CASE _diCmdState OF
	0://判断对应指令，是否已经处于完成状态，防止出现重复触发情况	
		_diCmdState := _diCmdState + 1;	
	1://传送力值和速度参数
		IF NOT _aRead_VAR.bExecute//等待最后接收结束
		THEN
			_tonDelay(IN:= TRUE,pt:=T#20MS);
			st_IOData.O_ClampForceSet := rTorqueSet;
			st_IOData.O_ClampSpeedSet := rSpeedSet;	
			st_IOData.O_ClampPosSet := rPosAngleSet;	
			IF _tonDelay.Q
			THEN	
				_aEnableSignal[1] := TRUE;//启动参数数据发送	
				_tonDelay(IN:= FALSE);
				_tonCmdTimeout(in:=FALSE);
				_tonTimeout(in:=FALSE);
				_diCmdState := _diCmdState+1; 
			END_IF
		END_IF		
	2://设置读取参数	
		_tonDelay(IN:= NOT _aEnableSignal[1],PT:=T#200MS);
		_tonCmdTimeout(IN:= _aEnableSignal[1],pt:=T#2S);
		IF _tonDelay.Q
		THEN
			_tonCmdTimeout(in:=FALSE);
			_tonCmdTimeout(in:=FALSE);
			_tonDelay(in:=FALSE);
			_diCmdState := 4; 
		END_IF	
		IF _iSendReceiveState = 999
		THEN
			eErrorID := ERG_20_ERROR.FLT_CLAMPCMD_TIMEOUT;		
			_diCmdState := 100;
		END_IF		
	4://设置读取反馈数据
		_tonCmdTimeout(in:=FALSE);
		_tonDelay(IN:= FALSE);	
		_aEnableSignal[4] := TRUE;//读取状态反馈信息 
		_diCmdState := _diCmdState +1;//转到等待夹取完成 	
	5://等到操作完成
		_tonTimeout(in:=TRUE,pt:=T#10S); 
		_tonCmdTimeout(IN:= TRUE,pt:=T#2S);		
		IF NOT _aEnableSignal[4] //等待读取数据完成
		THEN
			_tonDelay(IN:= TRUE,pt:=T#40MS);
			IF st_IOData.I_ClampState = 0 AND ABS(st_IOData.O_ClampPosSet - st_IOData.I_ClampCurrentPos) <= 0.03 AND //松开位置成功
			   eCmd = ERG_20_CMD.Cmd_Release	//松开指令
			THEN			
				_tonCmdTimeout(in:=FALSE);
				_tonTimeout(in:=FALSE);  
				_diCmdState := 100;
				xComplete := TRUE;
			END_IF		
			IF st_IOData.I_ClampState = 2 AND//夹住物体
				 eCmd = ERG_20_CMD.Cmd_Clamp	//夹紧指令
			THEN			
				_tonCmdTimeout(in:=FALSE);
				_tonTimeout(in:=FALSE);  
				_diCmdState := 100;
				xComplete := TRUE;
			END_IF				
			IF st_IOData.I_ClampState = 2 AND //松开位置的时候，检测是否堵转
       	 eCmd = ERG_20_CMD.Cmd_Release	//松开指令
			THEN	
  			_iNGCount := _iNGCount + 1;		
				IF _iNGCount <= 3
				THEN
				  _tonDelay(IN:=FALSE);
					_diCmdState := _diCmdState + 1;
				ELSE
					_tonCmdTimeout(in:=FALSE);
					_tonTimeout(in:=FALSE);  
					eErrorID := ERG_20_ERROR.FLT_ClAMP_RELEASEFAIL;		
					_diCmdState := 999;
				END_IF				
			END_IF		
			IF st_IOData.I_ClampState = 0 AND ABS(st_IOData.O_ClampPosSet - st_IOData.I_ClampCurrentPos) <= 0.03 AND//没有夹住物体，到位置，判定夹持失败(放个误差数值)
				 eCmd = ERG_20_CMD.Cmd_Clamp	//夹紧指令
			THEN
				_iNGCount := _iNGCount + 1;		
				IF _iNGCount <= 3
				THEN
				  _tonDelay(IN:=FALSE);
					_diCmdState := _diCmdState + 1;
				ELSE
					_tonCmdTimeout(in:=FALSE);
					_tonTimeout(in:=FALSE);  			
					eErrorID := ERG_20_ERROR.FLT_ClAMP_CLAMPFAIL;		
					_diCmdState := 999;
				END_IF
			END_IF	
			IF _tonDelay.Q//做延时刷新
			THEN
				_diCmdState := 4;
			END_IF			
		END_IF
		IF _iSendReceiveState = 999//回原点指令响应超时
		THEN
			eErrorID := ERG_20_ERROR.FLT_CLAMPCMD_TIMEOUT;		
			_diCmdState := 999;
		END_IF
		IF _tonTimeout.Q//回原点动作超时
		THEN
			eErrorID := ERG_20_ERROR.FLT_CLAMP_TIMEOUT;
			_diCmdState := 999;
		END_IF
	6:
		_tonDelay(IN:= TRUE,pt:=T#40MS);
		IF _tonDelay.Q//做延时刷新
		THEN			
			_diCmdState := 0;
		END_IF	
	ELSE
		;	
END_CASE
END_METHOD

METHOD CmdRotateAction
VAR_OUTPUT
	xComplete: BOOL;
END_VAR
// return the real actual fault number
IF eErrorID <> ERG_20_ERROR.NO_ERROR
THEN
  RETURN;  
END_IF
  
IF NOT xRefOk THEN//设备没有原点报警
	eErrorID := ERG_20_ERROR.FLT_xRefOk;
	RETURN;
END_IF

IF rTorqueSet>1 OR rTorqueSet<0.2
	OR rSpeedSet>1440 OR rSpeedSet<1
	OR rPosAngleSet>360000 OR rPosAngleSet<-360000
THEN
	eErrorID := ERG_20_ERROR.FLT_PARA;	
END_IF


CASE _diCmdState OF
	0://判断是否已经处于目标位置或者夹取完成状态，防止出现重复触发情况
		_diCmdState := _diCmdState + 1;
			diOldStep:=_diCmdState;
		_tonDelay(IN:= FALSE);
		IF eCmd = ERG_20_CMD.Cmd_RotateAbsRelease//只有绝对松瓶盖定位是有可能处于目标完成状态的，判断是否已经到目标位置
		THEN
			//检测是否已经处于目标位置
			IF ABS(rPosAngleSet - st_IOData.I_RotateCurrentPos) <= 0.03
			THEN
				_tonTimeout(in:=FALSE);  
				_diCmdState := 100;
				xComplete := TRUE;
			END_IF			
		END_IF
		IF eCmd = ERG_20_CMD.Cmd_RotateAbsClamp//只有绝对定位是有可能处于目标完成状态的，增量的是一定要动作的
		THEN
			//检测是否已经处于目标位置，要是到位置，代表夹紧失败，此时需要报警
			IF ABS(rPosAngleSet - st_IOData.I_RotateCurrentPos) <= 0.03
			THEN
				eErrorID := ERG_20_ERROR.FLT_ROTATE_CLAMPFAIL;
				_diCmdState := 999;
			END_IF
		END_IF
	1://传送参数
			diOldStep:=_diCmdState;
		IF NOT _aRead_VAR.bExecute//等待最后接收结束
		THEN
	    _tonDelay(IN:= TRUE,pt:=T#20MS);//保证执行的都是当次任务 			
			st_IOData.O_RotateForceSet := rTorqueSet;
			st_IOData.O_RotateSpeedSet := rSpeedSet;	
			st_IOData.O_RotatePosSet := rPosAngleSet;				
			IF _tonDelay.Q
			THEN				
				_aEnableSignal[2] := TRUE;//启动旋转绝对定位参数数据发送		    					
				_tonCmdTimeout(in:=FALSE);
				_tonDelay(IN:=FALSE);
				_diCmdState := _diCmdState+1; 	
			END_IF			
		END_IF	
	2://设置读取参数
			diOldStep:=_diCmdState;
		_tonDelay(IN:= NOT _aEnableSignal[2],PT:=T#200MS);//等待设备运行起来
		_tonCmdTimeout(IN:= _aEnableSignal[2],pt:=T#2S);
		IF _tonDelay.Q//等待电动夹爪开始响应
		THEN
			_tonTimeout(in:=FALSE);		
			_diCmdState := _diCmdState +1; 
		END_IF	
		IF _iSendReceiveState = 999//指令执行超时
		THEN
			eErrorID := ERG_20_ERROR.FLT_ROTATECMD_TIMEOUT;		
			_diCmdState := 999;
		END_IF	
	3://设置读取参数反馈
			diOldStep:=_diCmdState;
		_tonCmdTimeout(in:=FALSE);
		_tonDelay(IN:= FALSE);
	  _aEnableSignal[4] := TRUE;   
		_diCmdState := _diCmdState +1;//
	4:
		diOldStep:=_diCmdState;
		_tonTimeout(in:=TRUE,pt:=T#20S); 
		_tonCmdTimeout(IN:= TRUE,pt:=T#2S);
		//进行数据刷新		
		IF NOT _aEnableSignal[4] //等待读取数据完成
		THEN
			_tonDelay(IN:= TRUE,pt:=T#50MS);
			IF ( st_IOData.I_RotateState = 0 ) AND ABS(st_IOData.O_RotatePosSet - st_IOData.I_RotateCurrentPos) <= 0.03 AND //旋转是否到位置,只有在松开瓶盖的时候会有这种操作
				 ( eCmd = ERG_20_CMD.Cmd_RotateAbsRelease )
			THEN			
				_tonTimeout(in:=FALSE);  
				_diCmdState := 100;
				xComplete := TRUE;
			END_IF		 
			IF ( st_IOData.I_RotateState = 2 OR st_IOData.I_RotateState = 4 ) AND //旋转夹瓶盖处理，只有出现堵转（达到设置力反馈）
				 ( eCmd = ERG_20_CMD.Cmd_RotateAbsClamp )
			THEN			
				_tonTimeout(in:=FALSE);  
				_diCmdState := 100;
				xComplete := TRUE;
			END_IF			
			IF _tonDelay.Q//做刷新处理
			THEN
				_diCmdState := _diCmdState - 1;
			END_IF
		END_IF
		IF ( st_IOData.I_RotateState = 0 ) AND ABS(st_IOData.O_RotatePosSet - st_IOData.I_RotateCurrentPos) <= 0.03 AND //关盖打滑,直接到设置位置了
			 ( eCmd = ERG_20_CMD.Cmd_RotateAbsClamp )
		THEN	
			_tonDelay(IN:=FALSE);
			eErrorID := ERG_20_ERROR.FLT_ROTATE_CLAMPFAIL;
			_diCmdState := 999;
		END_IF
		IF ( st_IOData.I_RotateState = 2 OR st_IOData.I_RotateState = 4) AND //开盖失败，直接堵转，开不开瓶盖
			 ( eCmd = ERG_20_CMD.Cmd_RotateAbsRelease )
		THEN	
			_iNGCount := _iNGCount + 1;		
			IF _iNGCount <= 3//检测是否有正时报警发生
			THEN
				_tonDelay(IN:=FALSE);
				_diCmdState := _diCmdState + 1;
			ELSE
				eErrorID := ERG_20_ERROR.FLT_ROTATE_RELEASEFAIL;
				_diCmdState := 999;
			END_IF
		END_IF
		IF _iSendReceiveState = 999//回原点指令响应超时
		THEN
			eErrorID := ERG_20_ERROR.FLT_ROTATECMD_TIMEOUT;		
			_diCmdState := 999;
		END_IF
		IF _tonTimeout.Q//回原点动作超时
		THEN
			eErrorID := ERG_20_ERROR.FLT_ROTATE_TIMEOUT;
			_diCmdState := 999;
		END_IF
	5://报警再次确定
			diOldStep:=_diCmdState;
		_tonDelay(IN:= TRUE,pt:=T#40MS);
		IF _tonDelay.Q//做延时刷新
		THEN			
			_diCmdState := 0;
		END_IF		
	ELSE
		;	
END_CASE
END_METHOD

METHOD CmdRotateAction_Rel
VAR_OUTPUT
	xComplete: BOOL;
END_VAR
// return the real actual fault number
IF eErrorID <> ERG_20_ERROR.NO_ERROR
THEN
  RETURN;  
END_IF
  
IF NOT xRefOk THEN//设备没有原点报警
	eErrorID := ERG_20_ERROR.FLT_xRefOk;
	RETURN;
END_IF

IF rTorqueSet>1 OR rTorqueSet<0.2
	OR rSpeedSet>1440 OR rSpeedSet<1
	OR rPosAngleSet>36000 OR rPosAngleSet<-36000
THEN
	eErrorID := ERG_20_ERROR.FLT_PARA;	
END_IF

CASE _diCmdState OF
	0://判断是否已经处于目标位置或者夹取完成状态，防止出现重复触发情况
		_tonDelay(IN:= FALSE);
		IF NOT _aRead_VAR.bExecute THEN		
			_diCmdState := _diCmdState + 1;
			_rLastRotatePos:= st_IOData.I_RotateCurrentPos;
		END_IF	
	1://传送参数
		_tonDelay(IN:= TRUE,pt:=T#20MS);//保证执行的都是当次任务 			
		st_IOData.O_RotateForceSet := rTorqueSet;
		st_IOData.O_RotateSpeedSet := rSpeedSet;	
		st_IOData.O_RotatePosSet := rPosAngleSet;				
		IF _tonDelay.Q
		THEN				
			_aEnableSignal[3] := TRUE;//启动旋转绝对定位参数数据发送		    					
			_tonCmdTimeout(in:=FALSE);
			_tonDelay(IN:=FALSE);
			_diCmdState := _diCmdState+1; 	
		END_IF			
	2://设置读取参数
		_tonDelay(IN:= NOT _aEnableSignal[3],PT:=T#200MS);//等待设备运行起来
		_tonCmdTimeout(IN:= _aEnableSignal[3],pt:=T#2S);
		IF _tonDelay.Q//等待电动夹爪开始响应
		THEN
			_tonTimeout(in:=FALSE);		
			_diCmdState := _diCmdState +1; 
		END_IF	
		IF _iSendReceiveState = 999//指令执行超时
		THEN
			eErrorID := ERG_20_ERROR.FLT_ROTATECMD_TIMEOUT;		
			_diCmdState := 999;
		END_IF	
	3://设置读取参数反馈
		_tonCmdTimeout(in:=FALSE);
		_tonDelay(IN:= FALSE);
	  _aEnableSignal[4] := TRUE;   
		_diCmdState := _diCmdState +1;//
	4:
		_tonTimeout(in:=TRUE,pt:=T#20S); 
		_tonCmdTimeout(IN:= TRUE,pt:=T#2S);
		//进行数据刷新		
		IF NOT _aEnableSignal[4] //等待读取数据完成
		THEN
			_tonDelay(IN:= TRUE,pt:=T#50MS);
			IF ( st_IOData.I_RotateState = 0 ) 
					AND (st_IOData.I_RotateCurrentPos - _rLastRotatePos) <= rPosAngleSet+0.03 
					AND (st_IOData.I_RotateCurrentPos - _rLastRotatePos) >= rPosAngleSet-0.03 //旋转是否到位置,只有在松开瓶盖的时候会有这种操作
				 AND ( eCmd = ERG_20_CMD.Cmd_RotateRelRelease )
			THEN			
				_tonTimeout(in:=FALSE);  
				_diCmdState := 100;
				xComplete := TRUE;
			END_IF		 
			IF ( st_IOData.I_RotateState = 2 OR st_IOData.I_RotateState = 4 ) AND //旋转夹瓶盖处理，只有出现堵转（达到设置力反馈）
				 ( eCmd = ERG_20_CMD.Cmd_RotateRelClamp )
			THEN			
				_tonTimeout(in:=FALSE);  
				_diCmdState := 100;
				xComplete := TRUE;
			END_IF			
			IF _tonDelay.Q//做刷新处理
			THEN
				_diCmdState := _diCmdState - 1;
			END_IF
		END_IF
		
		IF ( st_IOData.I_RotateState = 0 )  
 				AND (st_IOData.I_RotateCurrentPos - _rLastRotatePos) <= rPosAngleSet+0.03 
				AND (st_IOData.I_RotateCurrentPos - _rLastRotatePos) >= rPosAngleSet-0.03  //关盖打滑,直接到设置位置了
			  AND( eCmd = ERG_20_CMD.Cmd_RotateRelClamp )
		THEN	
			_tonDelay(IN:=FALSE);
			eErrorID := ERG_20_ERROR.FLT_ROTATE_CLAMPFAIL;
			_diCmdState := 999;
		END_IF
		IF ( st_IOData.I_RotateState = 2 OR st_IOData.I_RotateState = 4) AND //开盖失败，直接堵转，开不开瓶盖
			 ( eCmd = ERG_20_CMD.Cmd_RotateRelRelease )
		THEN	
			_iNGCount := _iNGCount + 1;		
			IF _iNGCount <= 3//检测是否有正时报警发生
			THEN
				_tonDelay(IN:=FALSE);
				_diCmdState := _diCmdState + 1;
			ELSE
				eErrorID := ERG_20_ERROR.FLT_ROTATE_RELEASEFAIL;
				_diCmdState := 999;
			END_IF
		END_IF
		IF _iSendReceiveState = 999//回原点指令响应超时
		THEN
			eErrorID := ERG_20_ERROR.FLT_ROTATECMD_TIMEOUT;		
			_diCmdState := 999;
		END_IF
		IF _tonTimeout.Q//回原点动作超时
		THEN
			eErrorID := ERG_20_ERROR.FLT_ROTATE_TIMEOUT;
			_diCmdState := 999;
		END_IF
	5://报警再次确定
		_tonDelay(IN:= TRUE,pt:=T#40MS);
		IF _tonDelay.Q//做延时刷新
		THEN			
			_diCmdState := 3;
		END_IF		
	ELSE
		;	
END_CASE
END_METHOD

ACTION ConnectAction:
(**********************************调用收发功能块**********************************)
//状态反馈功能调用
_aRead_VAR(
	sIPAddr:= stPara.strSlaveIP, 
	nTCPPort:=stPara.iSlavePort , 
	nUnitID:= stPara.bySlaveID, 
	nQuantity:= 18, 
	nMBAddr:= 16#0040, 
	cbLength:= 36, 
	pDestAddr:= ADR(_aFeedbackData), 
	bExecute:= , 
	tTimeout:= T#1S, 
	bBusy=> , 
	bError=> , 
	nErrId=> , 
	cbRead=> );		
	
//指令控制部分	
_aWtirt_VAR[0](
	sIPAddr:= stPara.strSlaveIP,
	nTCPPort:= stPara.iSlavePort, 
	nUnitID:= stPara.bySlaveID, 
	nQuantity:= 1, 
	nMBAddr:= 16#0000, 
	cbLength:= 2, 
	pSrcAddr:= ADR(_aControlData[0,0]), 
	bExecute:= , 
	tTimeout:= T#1S, 
	bBusy=> , 
	bError=> , 
	nErrId=> );	
		
_aWtirt_VAR[1](
	sIPAddr:= stPara.strSlaveIP,
	nTCPPort:= stPara.iSlavePort, 
	nUnitID:= stPara.bySlaveID, 
	nQuantity:= 6, 
	nMBAddr:= 16#0002, 
	cbLength:= 12, 
	pSrcAddr:= ADR(_aControlData[1,0]), 
	bExecute:= , 
	tTimeout:= T#1S, 
	bBusy=> , 
	bError=> , 
	nErrId=> );		
	
_aWtirt_VAR[2](
	sIPAddr:= stPara.strSlaveIP,
	nTCPPort:= stPara.iSlavePort, 
	nUnitID:= stPara.bySlaveID, 
	nQuantity:= 8, 
	nMBAddr:= 16#000A, 
	cbLength:= 16, 
	pSrcAddr:= ADR(_aControlData[2,0]), 
	bExecute:= , 
	tTimeout:= T#1S, 
	bBusy=> , 
	bError=> , 
	nErrId=> );		
	
_aWtirt_VAR[3](
	sIPAddr:= stPara.strSlaveIP,
	nTCPPort:= stPara.iSlavePort, 
	nUnitID:= stPara.bySlaveID, 
	nQuantity:= 8, 
	nMBAddr:= 16#000E, 
	cbLength:= 16, 
	pSrcAddr:= ADR(_aControlData[3,0]), 
	bExecute:= , 
	tTimeout:= T#1S, 
	bBusy=> , 
	bError=> , 
	nErrId=> );	
	
//收发流程管控
CASE _iSendReceiveState OF 
	0:
		_tonDelay2(IN:= FALSE);
		_iChannelIndex:= -1;
		FOR i := 0 TO 5 BY 1//进行读取指令的轮训
		DO
		 IF _aEnableSignal[i]//检测有控制指令发生
		 THEN
			 _iChannelIndex:=i;    
			END_IF 
		END_FOR
		IF _iChannelIndex>=4//有读取反馈指令
		THEN								
			IF NOT _aRead_VAR.bBusy AND NOT _aRead_VAR.bError
			THEN
				_aRead_VAR(bExecute := _aEnableSignal[_iChannelIndex]);
				_iSendReceiveState := 10;	
			ELSIF 
				_aRead_VAR.bError
				THEN
				_iSendReceiveState := 999;												
			END_IF													
		END_IF			
		IF _iChannelIndex>=0 AND _iChannelIndex<=3//有控制触发指令
		THEN		
			IF  NOT _aWtirt_VAR[_iChannelIndex].bBusy AND NOT _aWtirt_VAR[_iChannelIndex].bError 
			THEN
				_aWtirt_VAR[_iChannelIndex](bExecute := _aEnableSignal[_iChannelIndex]);
				_iSendReceiveState := 10;							
			END_IF
		END_IF
		
	10://等待读取响应	
		_tonDelay2(IN:= TRUE,PT:=T#3S);
		IF _tonDelay2.Q//超时
		THEN
			_iSendReceiveState:= 999;					
		END_IF				
		IF _iChannelIndex>=4
		THEN					
			IF NOT _aRead_VAR.bBusy AND NOT _aRead_VAR.bError
			THEN
				_iComNGCount := 0;
				_aEnableSignal[_iChannelIndex] := FALSE;
				_aRead_VAR.bExecute := FALSE;
				_iSendReceiveState := 0;//等待下次触发
			END_IF
			IF _aRead_VAR.bError
			THEN
				_iComNGCount := _iComNGCount + 1;//错误次数加一
				IF _iComNGCount >= 3//重发多次失败
				THEN
					eOperErrorID := _aRead_VAR.nErrId;
					_aRead_VAR.bExecute := FALSE;
					_iSendReceiveState := 999;//进入错误发生状态
				ELSE
					_tonDelay1(in:=FALSE);
					_aRead_VAR.bExecute:= FALSE;
					_iSendReceiveState := _iSendReceiveState + 1;
				END_IF						
			END_IF			
		END_IF				
		IF _iChannelIndex>=0 AND _iChannelIndex<=3		
		THEN	
			IF NOT _aWtirt_VAR[_iChannelIndex].bBusy AND NOT _aWtirt_VAR[_iChannelIndex].bError
			THEN
				_iComNGCount := 0;
				_aEnableSignal[_iChannelIndex] := FALSE;
				_aWtirt_VAR[_iChannelIndex].bExecute := FALSE;
				_iSendReceiveState := 0;//等待下次触发
			END_IF
			IF _aWtirt_VAR[_iChannelIndex].bError
			THEN
				_iComNGCount := _iComNGCount + 1;//错误次数加一
				IF _iComNGCount >= 3//重发多次失败
				THEN
					eOperErrorID := _aWtirt_VAR[_iChannelIndex].nErrId;
					_aWtirt_VAR[_iChannelIndex].bExecute := FALSE;
					_iSendReceiveState := 999;//进入错误发生状态
				ELSE
					_tonDelay1(in:=FALSE);
					_aWtirt_VAR[_iChannelIndex].bExecute:= FALSE;
					_iSendReceiveState := _iSendReceiveState + 1;
				END_IF					
			END_IF				
		END_IF
	11://延时，进行补发操作
		_tonDelay1(in:=TRUE,pt:=T#300MS);				
		IF _tonDelay1.Q
		THEN		 
			_iSendReceiveState := 0;
		END_IF	
	999://错误状态，等待复位发生
		_xConnect_ERROR := TRUE;
		_tonDelay1(in:=NOT _tonDelay1.Q,pt:=T#20MS);
		_aRead_VAR(bExecute := _tonDelay1.Q);	
		_tonDelay3(pt:=T#100MS);	
		IF _tonDelay3.Q
		THEN			
			_xConnect_ERROR := FALSE;
			_iComNGCount := 0;			
			_iSendReceiveState := 0;//重新开始
			_aRead_VAR(bExecute := FALSE);	
			_tonDelay1(IN:=FALSE);
			_tonDelay3(IN:=FALSE);
		END_IF
		IF _fResetCheck.Q
		THEN
			_aWtirt_VAR[0](bExecute := FALSE);
			_aWtirt_VAR[1](bExecute := FALSE);
			_aWtirt_VAR[2](bExecute := FALSE);
			_aWtirt_VAR[3](bExecute := FALSE);			
			_aRead_VAR(bExecute := FALSE);	
			_tonDelay3.IN := TRUE;
		END_IF
	ELSE
		;
END_CASE
END_ACTION

METHOD CyclicAction
VAR_INPUT
END_VAR
VAR_OUTPUT
	xComplete: BOOL;
END_VAR
IF xAbort=0 THEN
    IF xFirstInvocation THEN
    (*
    * Staring
    * for then first (!) invocaion,
    * sample then input variables
    *)
			_xReadStatus := FALSE;
			_iCount := 0;
			_diCmdState := 0;
			_iNGCount := 0;
			xFirstInvocation:=0;	
			_aRead_VAR.bExecute:= false;		
    END_IF    
    REPEAT 				
		  (**************************检查是否有硬件报错(检测总线是否报错)**********************************) 			
			//下面几个报警需要断驱动器的电才能消除报警
			IF st_IOData.I_DeviceERRORState <> 0 
			THEN
				eErrorID := ERG_20_ERROR.FLT_DEVICE_ERROR;//过热报警
			END_IF	

			IF NOT xPowerHmi//驱动器没有上电
			THEN
				eERRORID := ERG_20_ERROR.FLT_POWERON;//需要检查硬件，硬件有问题
			END_IF
		
			//判断指令类型
			CASE eCmd OF
					ERG_20_CMD.Cmd_Clamp,ERG_20_CMD.Cmd_Release://执行夹爪指令	
            eClampActCmd := eCmd ;				
						CmdClampAction(xComplete=> xComplete);				
					ERG_20_CMD.Cmd_Org://执行回原点指令
						mCmdOrgAction(xComplete=> xComplete);
					ERG_20_CMD.Cmd_RotateAbsClamp,ERG_20_CMD.Cmd_RotateAbsRelease:
						CmdRotateAction(xComplete=> xComplete);
					ERG_20_CMD.Cmd_RotateRelClamp,ERG_20_CMD.Cmd_RotateRelRelease:
						CmdRotateAction_Rel(xComplete=> xComplete);												
					ELSE
						;	
				END_CASE  
      UNTIL (TRUE)
	END_REPEAT
END_IF


IF xAbort OR xComplete OR eErrorID<>ERG_20_ERROR.NO_ERROR THEN    
    (*
    * Cleaning
    * => free as much allocated resources as possible
    *)    
    tOperationTimer(IN:=0);
END_IF
END_METHOD

{attribute 'hide'}
METHOD PRIVATE FINAL HandleAbortedState
VAR_INPUT
END_VAR
VAR_OUTPUT
	xAgain: BOOL;
END_VAR
VAR
	xComplete: BOOL;
END_VAR
IF xAborted AND xResetRequest THEN
    eState:=STATE.RESETING;
    xAgain:=1;
ELSE
    xBusy:=0;
    xAborted:=1;
    //xResetRequest:=(xExecute=0);
    xAgain:=0;(* !!! *)
END_IF
END_METHOD

{attribute 'hide'}
METHOD PRIVATE FINAL HandleAbortingState
VAR_INPUT
END_VAR
VAR_OUTPUT
	xAgain: BOOL;
END_VAR
VAR
	xComplete: BOOL;
END_VAR
AbortAction(xComplete=> xComplete, eErrorID=> eErrorID);

IF eErrorID<>ERG_20_ERROR.NO_ERROR THEN
    eState:=STATE.INERROR;
    xAgain:=1;
ELSIF xComplete THEN
    eState:=STATE.ABORTED;
    xAgain:=1;
END_IF
END_METHOD

{attribute 'hide'}
METHOD PRIVATE FINAL HandleDoneState
VAR_INPUT
END_VAR
VAR_OUTPUT
	xAgain: BOOL;
END_VAR
//在运行过程中要是切换模式，再运行完成之后，检测到模式的切换，就需要回到初始位置，进行下一次执行准备
IF _xDone AND ((xExecute=0) OR ( _xModeChange AND NOT _xAutoOpe ) OR ( NOT xAutoMode AND NOT xDeviceRunning AND ( NOT _xAutoOpe OR _xHMIOpe))) THEN
	eState:=STATE.RESETING;
	xAgain:=1;
ELSE
	xBusy:=0;
	_xDone:=1;
	//xResetRequest:=(xExecute=0);
	xAgain:=0;(* !!! *)
END_IF
END_METHOD

{attribute 'hide'}
METHOD PRIVATE FINAL HandleDormantState
VAR_INPUT
END_VAR
VAR_OUTPUT
	xAgain: BOOL;
END_VAR

IF xExecute THEN
    xBusy:=1;
    eState:=STATE.EXECUTING;
    xAgain:=1;
END_IF


IF st_IOData.I_DeviceERRORState <> 0//检测硬件是否报错
THEN
	eERRORID := ERG_20_ERROR.FLT_DEVICE_ERROR;//需要检查硬件，硬件有问题
END_IF
IF NOT xPowerHmi//驱动器没有上电
THEN
	eERRORID := ERG_20_ERROR.FLT_POWERON;//需要检查硬件，硬件有问题
END_IF
	
IF _fResetCheck.Q//清空报警
THEN
	eERRORID := ERG_20_ERROR.No_ERROR;
END_IF
(********************************等待手动操作******************************)
//初始化指令
_rHMIInit(CLK:= xHMInitButton AND eErrorID = ERG_20_ERROR.NO_ERROR AND NOT xAutoMode AND NOT xDeviceRunning );
_rInit(CLK:= xInitControl AND eErrorID = ERG_20_ERROR.NO_ERROR AND ( xAutoMode OR  xDeviceRunning ));
IF _rHMIInit.Q OR _rInit.Q
THEN
	eCmd := ERG_20_CMD.Cmd_Org;
	xExecute := TRUE;
END_IF
//轮询
FOR ii := 1 TO 5 BY 1
DO 
	//夹紧轴夹紧控制
	_rHMIClamp[ii](CLK:= aHMIClampButton[ii] AND eErrorID = ERG_20_ERROR.NO_ERROR AND NOT xAutoMode AND NOT xDeviceRunning );
	_rClamp[ii](CLK:= aClampControl[ii] AND eErrorID = ERG_20_ERROR.NO_ERROR AND ( xAutoMode OR xDeviceRunning ) );
	IF _rHMIClamp[ii].Q OR _rClamp[ii].Q
	THEN
		rTorqueSet := aHMIClampPara[ii].rTorqueSet;
		rSpeedSet := aHMIClampPara[ii].rSpeedSet;
		rPosAngleSet := aHMIClampPara[ii].rPosAngleSet;
		eCmd := ERG_20_CMD.Cmd_Clamp;
		xExecute := TRUE;
	END_IF	
	//夹紧轴松开指令
	_rHMIRelease[ii](CLK:= aHMIReleaseButton[ii] AND eErrorID = ERG_20_ERROR.NO_ERROR AND NOT xAutoMode AND NOT xDeviceRunning );
	_rRelease[ii](CLK:= aReleaseControl[ii] AND eErrorID = ERG_20_ERROR.NO_ERROR AND ( xAutoMode OR  xDeviceRunning ));
	IF _rHMIRelease[ii].Q OR _rRelease[ii].Q
	THEN
		rTorqueSet := aHMIReleasePara[ii].rTorqueSet;
		rSpeedSet := aHMIReleasePara[ii].rSpeedSet;
		rPosAngleSet := aHMIReleasePara[ii].rPosAngleSet;
		eCmd := ERG_20_CMD.Cmd_Release;
		xExecute := TRUE;
	END_IF		
  //旋转轴关盖控制
	_rHMIRotateClamp[ii](CLK:= aHMIRotateClampButton[ii] AND eErrorID = ERG_20_ERROR.NO_ERROR AND NOT xAutoMode AND NOT xDeviceRunning );
	_rRotateClamp[ii](CLK:= aRotateClampControl[ii] AND eErrorID = ERG_20_ERROR.NO_ERROR AND ( xAutoMode OR xDeviceRunning ) );
	IF _rHMIRotateClamp[ii].Q OR _rRotateClamp[ii].Q
	THEN
		rTorqueSet := aHMIRotateClampPara[ii].rTorqueSet;
		rSpeedSet := aHMIRotateClampPara[ii].rSpeedSet;
		rPosAngleSet := aHMIRotateClampPara[ii].rPosAngleSet;
		eCmd := ERG_20_CMD.Cmd_RotateAbsClamp;
		xExecute := TRUE;
	END_IF	
	//旋转轴松盖指令
	_rHMIRotateRelease[ii](CLK:= aHMIRotateReleaseButton[ii] AND eErrorID = ERG_20_ERROR.NO_ERROR AND NOT xAutoMode AND NOT xDeviceRunning );
	_rRotateRelease[ii](CLK:= aRotateReleaseControl[ii] AND eErrorID = ERG_20_ERROR.NO_ERROR AND ( xAutoMode OR  xDeviceRunning ));
	IF _rHMIRotateRelease[ii].Q OR _rRotateRelease[ii].Q
	THEN
		rTorqueSet := aHMIRotateReleasePara[ii].rTorqueSet;
		rSpeedSet := aHMIRotateReleasePara[ii].rSpeedSet;
		rPosAngleSet := aHMIRotateReleasePara[ii].rPosAngleSet;
		eCmd := ERG_20_CMD.Cmd_RotateAbsRelease;
		xExecute := TRUE;
	END_IF		
  //旋转轴关盖控制
	_rHMIRotateRelClamp[ii](CLK:= aHMIRotateClampRelButton[ii] AND eErrorID = ERG_20_ERROR.NO_ERROR AND NOT xAutoMode AND NOT xDeviceRunning );
	_rRotateRelClamp[ii](CLK:= aRotateClampRelControl[ii] AND eErrorID = ERG_20_ERROR.NO_ERROR AND ( xAutoMode OR xDeviceRunning ) );
	IF _rHMIRotateRelClamp[ii].Q OR _rRotateRelClamp[ii].Q
	THEN
		rTorqueSet := aHMIRotateClampRelPara[ii].rTorqueSet;
		rSpeedSet := aHMIRotateClampRelPara[ii].rSpeedSet;
		rPosAngleSet := aHMIRotateClampRelPara[ii].rPosAngleSet;
		eCmd := ERG_20_CMD.Cmd_RotateRelClamp;
		xExecute := TRUE;
	END_IF	
	//旋转轴松盖指令
	_rHMIRotateRelRelease[ii](CLK:= aHMIRotateReleaseRelButton[ii] AND eErrorID = ERG_20_ERROR.NO_ERROR AND NOT xAutoMode AND NOT xDeviceRunning );
	_rRotateRelRelease[ii](CLK:= aRotateReleaseRelControl[ii] AND eErrorID = ERG_20_ERROR.NO_ERROR AND ( xAutoMode OR  xDeviceRunning ));
	IF _rHMIRotateRelRelease[ii].Q OR _rRotateRelRelease[ii].Q
	THEN
		rTorqueSet := aHMIRotateReleaseRelPara[ii].rTorqueSet;
		rSpeedSet := aHMIRotateReleaseRelPara[ii].rSpeedSet;
		rPosAngleSet := aHMIRotateReleaseRelPara[ii].rPosAngleSet;
		eCmd := ERG_20_CMD.Cmd_RotateRelRelease;
		xExecute := TRUE;
	END_IF
END_FOR
END_METHOD

{attribute 'hide'}
METHOD PRIVATE FINAL  HandleErrorState
VAR_INPUT
END_VAR
VAR_OUTPUT
	xAgain: BOOL;
END_VAR
IF xError THEN
	IF eErrorID < ERG_20_ERROR.FLT_ClAMP_CLAMPFAIL//正常执行报警
	THEN
		IF xResetRequest OR NOT xExecute//按照正常逻辑进行处理复位处理就可以
		THEN
				eState:=STATE.RESETING;
				xAgain:=1;
		END_IF
	ELSE//操作失败报警（有可能需要进行程序跳步处理，此时，在自动模式下不允许被复位掉，防止，程序异常死机）
		IF ( NOT xAutoMode AND xDeviceRunning ) OR xAutoMode
		THEN 
			IF NOT xExecute//按照正常逻辑进行处理复位处理就可以
			THEN 
				eState:=STATE.RESETING;
				xAgain:=1;
			END_IF
		ELSE
			IF xResetRequest OR NOT xExecute//按照正常逻辑进行处理复位处理就可以
			THEN
				eState:=STATE.RESETING;
				xAgain:=1;
			END_IF
		END_IF
	END_IF
ELSE
	xBusy:=0;
	xError:=1;    
	xAgain:=0;(* !!! *)
END_IF
END_METHOD

{attribute 'hide'}
METHOD PRIVATE FINAL HandleExecutingState
VAR_INPUT
END_VAR
VAR_OUTPUT
	xAgain: BOOL;
END_VAR
VAR
	xComplete: BOOL;
END_VAR
IF xAbort=0 THEN   
    CyclicAction(xComplete=> xComplete);
END_IF

IF eErrorID<>ERG_20_ERROR.NO_ERROR THEN
    eState:=STATE.INERROR;
    xAgain:=1;
ELSIF xAbort THEN
    eState:=STATE.ABORTING;
    xAgain:=1;
ELSIF xComplete THEN
    eState:=STATE.DONE;
    xAgain:=1;
END_IF
END_METHOD

{attribute 'hide'}
METHOD PRIVATE FINAL HandleResettingState
VAR_INPUT
END_VAR
VAR_OUTPUT
	xAgain: BOOL;
END_VAR
VAR
	xComplete: BOOL;
END_VAR
ResetAction(xComplete=> xComplete);

IF xComplete THEN
		xExecute:=0;//清除输入指令 
    xBusy:=0;
    _xDone:=0;
    xError:=0;
    xAborted:=0;
    eErrorID:=ERG_20_ERROR.NO_ERROR;
    eState:=STATE.DORMANT;
    xFirstInvocation:=1;
    xAgain:=0;(* !!! *)
END_IF
END_METHOD

METHOD mCmdOrgAction
VAR_OUTPUT
	xComplete: BOOL;
END_VAR
// return the real actual fault number
IF eErrorID <> ERG_20_ERROR.NO_ERROR
THEN
  RETURN;  
END_IF

CASE _diCmdState OF
	0://a相关数据初始化
		IF NOT _aRead_VAR.bExecute//等待接收结束
		THEN			
			xRefOk := FALSE;//因为需要重新初始化，所以需要清除回原点完成标志位	
			_aFeedbackData[0]:=0;    
			_diCmdState := _diCmdState+1;						
		END_IF
	1://首次初始化写入参数
			_tonDelay(in:=FALSE);
			_tonCmdTimeout(in:=FALSE);
			_diCmdState:= 2;		
	2://a相关数据初始化
		IF NOT _aRead_VAR.bExecute//等待接收结束
		THEN
			_tonDelay(IN:= TRUE,pt:=T#20MS);
			st_IOData.O_Init := 1;//触发回原点指令
			IF _tonDelay.Q//错开刷新时序
			THEN
				_aEnableSignal[0] := TRUE;//启动数据发送	  
				_tonTimeout(in:=FALSE);    
				_diCmdState := _diCmdState+1;
			END_IF			
		END_IF	
	3://检测指令是否超时
		_tonDelay(IN:= NOT _aEnableSignal[0],PT:=T#200MS);
		_tonCmdTimeout(IN:= _aEnableSignal[0],pt:=T#2S);
		IF _tonDelay.Q
		THEN
			_tonCmdTimeout(in:=FALSE);
			_tonDelay(in:=FALSE);
			_diCmdState := _diCmdState+1; 
		END_IF	
		IF _iSendReceiveState = 999
		THEN
			eErrorID := ERG_20_ERROR.FLT_ORGCMD_TIMEOUT;		
			_diCmdState := 999;
		END_IF		
	4://设置读取数据反馈	 
		_tonCmdTimeout(in:=FALSE);
		_tonTimeout(in:=TRUE,pt:=T#10S); 
		_tonDelay(IN:= FALSE);
		_aEnableSignal[4]:= TRUE;//读取状态信息
		_diCmdState := _diCmdState +1; 
	5://等待数据接收完成		
		_tonTimeout(in:=TRUE,pt:=T#10S); 
		_tonCmdTimeout(IN:= TRUE,pt:=T#2S);
		IF NOT _aEnableSignal[4]//等待电动夹爪响应 
		THEN
			_tonDelay(IN:= TRUE,pt:=T#40MS);
			IF st_IOData.I_ClampInit = 5  //判断是否初始化成功
			THEN
				_tonCmdTimeout(in:=FALSE);
				_tonDelay(IN:= FALSE);
				_tonTimeout(in:=FALSE);  
				_diCmdState := 100;
				xRefOk := TRUE;//标记回原点成功
				xComplete := 1;
			END_IF
			IF _tonDelay.Q
			THEN
				_diCmdState := 4;
			END_IF
		END_IF
		IF _iSendReceiveState = 999//回原点指令响应超时
		THEN
			eErrorID := ERG_20_ERROR.FLT_ORGCMD_TIMEOUT;		
			_diCmdState := 999;
		END_IF
		IF _tonTimeout.Q//回原点动作超时
		THEN
			eErrorID := ERG_20_ERROR.FLT_ORG_TIMEOUT;
			_diCmdState := 999;
		END_IF			
	ELSE
		;
END_CASE
END_METHOD

{attribute 'hide'}
METHOD ResetAction
VAR_INPUT
END_VAR
VAR_OUTPUT
	xComplete: BOOL;
END_VAR
(*
* Cleaning
* => free all allocated resources
* => reinitialize instance variables
*)
tOperationTimer(IN:=0);

// init command state
_diCmdState := 0;
_tonCmdTimeout(in:=FALSE);
_tonTimeout(in:=FALSE);
_tonDelay(IN:=FALSE);
_xModeChange := FALSE;
_iNGCount := 0;
_xReadStatus := TRUE;//操作完成之后，默认开始群进行读取操作

//清除触发标志位
FOR i:= 0 TO 4 BY 1
DO
	_aEnableSignal[i] := FALSE;
END_FOR

xHMInitButton:=FALSE;	
xInitControl:=FALSE;
FOR i:=1 TO 5 BY 1
DO
	aHMIClampButton[i]:=FALSE;
	aHMIReleaseButton[i]:=FALSE;
	aClampControl[i]:=FALSE;
	aReleaseControl[i]:=FALSE;
	aHMIRotateClampButton[i]:=FALSE;
	aHMIRotateReleaseButton[i]:=FALSE;
	aRotateClampControl[i]:=FALSE;
	aRotateReleaseControl[i]:=FALSE;
	
	aHMIRotateClampRelButton[i]:=FALSE;
	aHMIRotateReleaseRelButton[i]:=FALSE;
	aRotateClampRelControl[i]:=FALSE;
	aRotateReleaseRelControl[i]:=FALSE;
END_FOR

xComplete:=1;
END_METHOD

END_FUNCTION_BLOCK

// ---- POUs/003_FB/0014_HITBOT/FB_ERG_20C.TcPOU
FUNCTION_BLOCK FB_ERG_20C EXTENDS FB_Modbus_Tcp
(*
********************************************************************************
* Name: FB_ERG_20C
*
* Author:  Automanh
* Version: 1.0.0
*
* Description:
*  HITBOT's Z_ERG_20C AutoClamp of Rotate and Holding
*  
*
* Remarks:
*
* Revisions:
*   1.0.0 -AutomanH Rebuild
*********************************************************************************)
VAR_INPUT
	xIReset:BOOL;
	xIManualMode:BOOL;
	xIAutoMode:BOOL;
	xIDeviceRunning:BOOL;
	xITryRun:BOOL;//空跑
	LocalClient:stModbusPara;
	stRunPara	:stSetPara;//运行参数	
	stDeviceOpe	:stOper_Para;//操作按钮
END_VAR
VAR_OUTPUT
	stDevice:stDeviceStatus;
	stPara:stDeviceStatus;
	stReadPara:stReadPara;
	iQErrorID:INT;
	strQErrorID:STRING;
END_VAR
VAR
	// 按钮输入
	OperR_TRIG: ARRAY[1..40] OF  R_TRIG;
	//本地参数
	stLocalPara:stHIBOTLocalPara;
	//操作指令
	iOperType:INT;
	// 循环用
	i: INT;
	// //操作类型计数
	iOperCounter: INT;
	// 步骤
	iRunStep,iOldRunStep: INT;
	iParaStep,iOldParaStep:INT;
	// 临时变量
	arwSetData: ARRAY[1..2] OF WORD;
	// 超时定时器
	tTimeout: ARRAY[1..5] OF TON;
	rTempData:REAL;//临时
END_VAR

MEMCPY(ADR(SUPER^.stModbusPara),ADR(LocalClient),SIZEOF(localClient));
SUPER^.M_Modbus();
ACT_Operation();
ACT_Running();
ACT_ERROR();
ACT_Reset();

ACTION ACT_ERROR:
tTimeout[1](IN:= iParaStep =iOldParaStep AND iParaStep<>0 , PT:= T#15S, Q=> , ET=> );
tTimeout[2](IN:= iRunStep =iOldRunStep AND iRunStep<>0 , PT:= T#15S, Q=> , ET=> );
IF		tTimeout[1].Q THEN
	  	stPara.xQError:=TRUE;
	  	stPara.xQBusy:=FALSE;
			iQErrorID:=HITBOT_ERROR.FLT_CMD_TIMEOUT;
	    iParaStep := 999;
END_IF

IF		tTimeout[2].Q THEN
			stDevice.xQError:=TRUE;
			stDevice.xQBusy:=FALSE;
			iQErrorID:=HITBOT_ERROR.FLT_CMD_TIMEOUT;
			iRunStep := 999;
END_IF

IF  iQErrorID<> HITBOT_ERROR.NO_ERROR  THEN
		stDevice.xQError:=TRUE;
END_IF
//报错内容输出
CASE iQErrorID OF 
		 HITBOT_ERROR.No_ERROR:
			 strQErrorID:='NO ERROR';
		 HITBOT_ERROR.FLT_PARA:
			 strQErrorID:='FLT_PARA';
		 HITBOT_ERROR.FLT_READ_PARA:
			 strQErrorID:='FLT_READ_PARA';
		 HITBOT_ERROR.FLT_SET_PARA:
			 strQErrorID:='FLT_SET_PARA';	
		 HITBOT_ERROR.FLT_CMD_TIMEOUT:
			 strQErrorID:='FLT_CMD_TIMEOUT';	
		 HITBOT_ERROR.FLT_RUN_ERROR:
			 strQErrorID:='FLT_RUN_ERROR';	
		 HITBOT_ERROR.FLT_CONFIGURE_PARA:
			 strQErrorID:='FLT_CONFIGURE_PARA';		
		 HITBOT_ERROR.FLT_NEED_INIT:
			 strQErrorID:='FLT_NEED_INIT';	
		 HITBOT_ERROR.FLT_CLAMP_EMPTY:
			strQErrorID:='FLT_CLAMP_EMPTY';		
END_CASE
END_ACTION

ACTION ACT_Operation:
FOR i:=1 TO 5 BY 1 DO
		OperR_TRIG[i](CLK:= (xIManualMode AND  stDeviceOpe.aHMIClampButton[i]) OR((xIAutoMode OR  xIDeviceRunning) AND stDeviceOpe.aClampControl[i]) , Q=> );	//夹紧
END_FOR
FOR i:=6 TO 10 BY 1DO
		OperR_TRIG[i](CLK:= (xIManualMode AND  stDeviceOpe.aHMIReleaseButton[i-5]) OR((xIAutoMode OR  xIDeviceRunning) AND stDeviceOpe.aReleaseControl[i-5]) , Q=> );	//松开
END_FOR
FOR i:=11 TO 15 BY 1 DO
		OperR_TRIG[i](CLK:= (xIManualMode AND  stDeviceOpe.aHMIRotateClampButton[i-10]) OR((xIAutoMode OR  xIDeviceRunning) AND stDeviceOpe.aRotateClampControl[i-10]) , Q=> );	//旋转拧紧
END_FOR

FOR i:=16 TO 20 BY 1 DO
		OperR_TRIG[i](CLK:= (xIManualMode AND  stDeviceOpe.aHMIRotateReleaseButton[i-15]) OR((xIAutoMode OR  xIDeviceRunning) AND stDeviceOpe.aRotateReleaseControl[i-15]) , Q=> );	//旋转松开
END_FOR

FOR i:=21 TO 25 BY 1 DO
		OperR_TRIG[i](CLK:= (xIManualMode AND  stDeviceOpe.aHMIRotateClampRelButton[i-20]) OR((xIAutoMode OR  xIDeviceRunning) AND stDeviceOpe.aRotateClampRelControl[i-20]) , Q=> );	//旋转拧紧-相对
END_FOR

FOR i:=26 TO 30 BY 1 DO
		OperR_TRIG[i](CLK:= (xIManualMode AND  stDeviceOpe.aHMIRotateReleaseRelButton[i-25]) OR((xIAutoMode OR  xIDeviceRunning) AND stDeviceOpe.aRotateReleaseRelControl[i-25]) , Q=> );	//旋转松开-相对
END_FOR
OperR_TRIG[31](CLK:= (xIManualMode AND  stDeviceOpe.xHMInitButton) OR((xIAutoMode OR  xIDeviceRunning) AND stDeviceOpe.xInitControl) , Q=> );	//初始化

FOR  i:= 1 TO 40 BY 1 DO
 	IF   OperR_TRIG[i].Q THEN
				iOperCounter:= i;
				stDevice.xQStart:=TRUE;
				EXIT;
	END_IF
END_FOR
//夹紧
FOR  i:=1 TO 5 BY 1 DO
 		IF   iOperCounter =i THEN
		 		stLocalPara.stClampPara.rPositionSet:=stRunPara.aHMIClampPara[i].rPositionSet;
				stLocalPara.stClampPara.rSpeedSet:=stRunPara.aHMIClampPara[i].rSpeedSet;
				stLocalPara.stClampPara.rCurrentSet:=stRunPara.aHMIClampPara[i].rCurrentSet;
				iOperType:=stCmdType.iClamp;
		END_IF
END_FOR
//松开
FOR  i:=6 TO 10 BY 1 DO
		IF   iOperCounter =i THEN
		 		stLocalPara.stClampPara.rPositionSet:=stRunPara.aHMIReleasePara[i-5].rPositionSet;
				stLocalPara.stClampPara.rSpeedSet:=stRunPara.aHMIReleasePara[i-5].rSpeedSet;
				stLocalPara.stClampPara.rCurrentSet:=stRunPara.aHMIReleasePara[i-5].rCurrentSet;
				iOperType:=stCmdType.iRelease;
		END_IF
END_FOR 
 //拧紧
FOR  i:=11 TO 15 BY 1 DO
 		IF   iOperCounter =i THEN
		 		stLocalPara.stRotateClampPara.rPositionSet:=stRunPara.aHMIRotateClampPara[i-10].rPositionSet;
				stLocalPara.stRotateClampPara.rSpeedSet:=stRunPara.aHMIRotateClampPara[i-10].rSpeedSet;
				stLocalPara.stRotateClampPara.rCurrentSet:=stRunPara.aHMIRotateClampPara[i-10].rCurrentSet;
				iOperType:=stCmdType.iRotateClamp;
		END_IF
END_FOR
//拧松
FOR  i:=16 TO 20 BY 1 DO
		IF   iOperCounter =i THEN
		 		stLocalPara.stRotateClampPara.rPositionSet:=stRunPara.aHMIRotateReleasePara[i-15].rPositionSet;
				stLocalPara.stRotateClampPara.rSpeedSet:=stRunPara.aHMIRotateReleasePara[i-15].rSpeedSet;
				stLocalPara.stRotateClampPara.rCurrentSet:=stRunPara.aHMIRotateReleasePara[i-15].rCurrentSet;
				iOperType:=stCmdType.iRotateRelease;
		END_IF
END_FOR 
 //相对拧紧
FOR  i:=21 TO 26 BY 1 DO
 		IF   iOperCounter =i THEN
		 		stLocalPara.stRotateClampPara.rPositionSet:=stRunPara.aHMIRotateRelClampPara[i-20].rPositionSet;
				stLocalPara.stRotateClampPara.rSpeedSet:=stRunPara.aHMIRotateRelClampPara[i-20].rSpeedSet;
				stLocalPara.stRotateRelAngle:=stRunPara.aHMIRotateRelClampPara[i-20].rCurrentSet;
				iOperType:=stCmdType.iRotateRelClamp;
		END_IF
END_FOR
//相对拧松
FOR  i:=26 TO 30 BY 1 DO
		IF   iOperCounter =i THEN
		 		stLocalPara.stRotateClampPara.rPositionSet:=stRunPara.aHMIRotateRelReleasePara[i-25].rPositionSet;
				stLocalPara.stRotateClampPara.rSpeedSet:=stRunPara.aHMIRotateRelReleasePara[i-25].rSpeedSet;
				stLocalPara.stRotateRelAngle:=stRunPara.aHMIRotateRelReleasePara[i-25].rCurrentSet;
				iOperType:=stCmdType.iRotateRelRelease;
		END_IF
END_FOR 

	IF   iOperCounter =31 THEN
				iOperType:=stCmdType.iInit;
	END_IF


MEMSET(ADR(stDeviceOpe),0,SIZEOF(stDeviceOpe));
END_ACTION

ACTION ACT_Para_Clamp:
CASE iParaStep OF	
	0://开始
			IF   stPara.xQStart THEN
			 		 stPara.xQStart:=FALSE;
					 stPara.xQBusy:=TRUE;
					 stPara.xQDone:=FALSE;
					  iParaStep := iParaStep + 1;
			 END_IF
 	1://查看夹爪电流，转速，转矩
			iOldParaStep:=iParaStep;
			IF 	(stLocalPara.stClampPara.rSpeedSet >=1  	AND 
			 		stLocalPara.stClampPara.rSpeedSet <=1000  )	AND
					(stLocalPara.stClampPara.rPositionSet >=0  AND 
					 stLocalPara.stClampPara.rPositionSet <= 20  )AND 
					(stLocalPara.stClampPara.rCurrentSet >=0.1  AND 
					 stLocalPara.stClampPara.rCurrentSet <=0.5  ) THEN
						iParaStep := iParaStep + 1;	
			ELSE
			 				iQErrorID :=HITBOT_ERROR.FLT_PARA;		
							iParaStep := 999;
			END_IF
	2://读取夹持速度和夹持电流
			iOldParaStep:=iParaStep;
			wMBAddReadRegs:=16#0004;
			wQuantityReadRegs:=4;
			xReadRegs:=TRUE;
			IF  fbReadRegs.bBusy THEN
			 	xReadRegs:=FALSE;
				iParaStep:=iParaStep+1;
			END_IF
	3://等待读取完成
			 	iOldParaStep:=iParaStep;
	  	  IF  NOT 	fbReadRegs.bBusy AND  NOT  	fbReadRegs.bError THEN
				 				//夹持速度
				
								stReadPara.rClampSpeed:=M_Little_Endian(pInputData:=ADR(arwDataReadRegs[1]));
								//夹持电流
						
								stReadPara.rClampCurrent:=M_Little_Endian(pInputData:=ADR(arwDataReadRegs[3]));
	  		 				 iParaStep:=iParaStep+1;
	  		 ELSIF   	fbReadRegs.bError THEN
	  		 			iParaStep:=999;				
	  		 			iQErrorID:=HITBOT_ERROR.FLT_READ_PARA;					
	  		 END_IF	
	4://夹持速度
				iOldParaStep:=iParaStep;
				IF stLocalPara.stClampPara.rSpeedSet <> stReadPara.rClampPosition THEN 
					 iParaStep:=iParaStep + 1;	
				ELSE
					 iParaStep:=iParaStep +4;
				END_IF
	5://夹持速度赋值
			iOldParaStep:=iParaStep;
			MEMCPY(ADR(arwSetData[1]),ADR(stLocalPara.stClampPara.rSpeedSet),SIZEOF(stLocalPara.stClampPara.rSpeedSet) ); 
			arwDataWriteRegs[1]:=arwSetData[2];
			arwDataWriteRegs[2]:=arwSetData[1];
			iParaStep:=iParaStep +1;
	6://夹持速度写入
			 iOldParaStep:=iParaStep;
			 wQuantityWriteRegs:=2;
			 wMBAddWriteRegs:=16#0004;
			 xWriteRegs:=TRUE;
			 IF  fbWriteRegs.bBusy THEN
					 xWriteRegs:=FALSE;
					 iParaStep:=iParaStep+1;
			END_IF	
	7://等待设定完成
				iOldParaStep:=iParaStep;
			 IF  NOT 	fbWriteRegs.bBusy AND  NOT fbWriteRegs.bError THEN
							  iParaStep:=iParaStep +1;
				ELSIF   	fbReadRegs.bError THEN
						 iParaStep:=999;				
						 iQErrorID:=HITBOT_ERROR.FLT_SET_PARA;					
				END_IF	
	8://夹持电流比较
				iOldParaStep:=iParaStep;
				IF stLocalPara.stClampPara.rCurrentSet <> stReadPara.rClampCurrent THEN 
					 iParaStep:=iParaStep + 1;	
				ELSE
					 iParaStep:=iParaStep + 4;
				END_IF
	9://夹持电流赋值
			iOldParaStep:=iParaStep;
			MEMCPY(ADR(arwSetData[1]),ADR(stLocalPara.stClampPara.rCurrentSet),SIZEOF(stLocalPara.stClampPara.rCurrentSet) ); 
			arwDataWriteRegs[1]:=arwSetData[2];
			arwDataWriteRegs[2]:=arwSetData[1];
			iParaStep:=iParaStep +1;
	10://夹持电流写入
			 iOldParaStep:=iParaStep;
			 wQuantityWriteRegs:=2;
			 wMBAddWriteRegs:=16#0006;
			 xWriteRegs:=TRUE;
			 IF  fbWriteRegs.bBusy THEN
					 xWriteRegs:=FALSE;
					 iParaStep:=iParaStep+1;
			END_IF	
	11://等待设定完成
				iOldParaStep:=iParaStep;
			 IF  NOT 	fbWriteRegs.bBusy AND  NOT fbWriteRegs.bError THEN
							  iParaStep:=iParaStep +1;
				ELSIF   	fbReadRegs.bError THEN
						 iParaStep:=999;				
						 iQErrorID:=HITBOT_ERROR.FLT_SET_PARA;					
				END_IF	
	12://写入电机使能
			iOldParaStep:=iParaStep;
			arwDataWriteRegs[1]:=1;
			iParaStep:=iParaStep +1;
	13://开始写入
			 iOldParaStep:=iParaStep;
			 wQuantityWriteRegs:=1;
			 wMBAddWriteRegs:=16#0016;
			 xWriteRegs:=TRUE;
			 IF  fbWriteRegs.bBusy THEN
					 xWriteRegs:=FALSE;
					 iParaStep:=iParaStep+1;
			END_IF	
	14://等待设定完成
				iOldParaStep:=iParaStep;
			 IF  NOT 	fbWriteRegs.bBusy AND  NOT fbWriteRegs.bError THEN
							  iParaStep:=100;
				ELSIF   	fbReadRegs.bError THEN
						 iParaStep:=999;				
						 iQErrorID:=HITBOT_ERROR.FLT_SET_PARA;					
				END_IF	
	100://参数写入完成
				iOldParaStep:=iParaStep;
				iOperType:=stOperType.iWait;
				stPara.xQBusy:=FALSE;
				stPara.xQDone:=TRUE;
				iParaStep:=0;		
	ELSE
		;	
END_CASE
END_ACTION

ACTION ACT_Para_Rotate:
CASE iParaStep OF	
	0://开始
			IF   stPara.xQStart THEN
			 		 stPara.xQStart:=FALSE;
					 stPara.xQBusy:=TRUE;
					 stPara.xQDone:=FALSE;
					  iParaStep := iParaStep + 1;
			 END_IF
 	1://查看夹爪电流，转速，角度
			iOldParaStep:=iParaStep;
			IF 	(	stLocalPara.stRotateClampPara.rSpeedSet >=1 	AND 
			 		stLocalPara.stRotateClampPara.rSpeedSet <=1080  )	AND
					(stLocalPara.stRotateClampPara.rPositionSet >=-3600000 AND 
					 stLocalPara.stRotateClampPara.rPositionSet <= 3600000 )AND 
					(stLocalPara.stRotateClampPara.rCurrentSet >=0.2  AND 
					 stLocalPara.stRotateClampPara.rCurrentSet <=1  ) THEN
						iParaStep := iParaStep + 1;	
			ELSE
			 				iQErrorID :=HITBOT_ERROR.FLT_PARA;		
							iParaStep := 999;
			END_IF
	2://读取旋转速度和旋转电流
			iOldParaStep:=iParaStep;
			wMBAddReadRegs:=16#000E;
			wQuantityReadRegs:=4;
			xReadRegs:=TRUE;
			IF  fbReadRegs.bBusy THEN
			 	xReadRegs:=FALSE;
				iParaStep:=iParaStep+1;
			END_IF
	3://等待读取完成
			 	iOldParaStep:=iParaStep;
	  	  IF  NOT 	fbReadRegs.bBusy AND  NOT  	fbReadRegs.bError THEN
								//旋转速度
								stReadPara.rRotateSpeed:=M_Little_Endian(pInputData:=ADR(arwDataReadRegs[1]));
								//旋转电流
								stReadPara.rRotateCurrent:=M_Little_Endian(pInputData:=ADR(arwDataReadRegs[3]));
	
	  		 				 iParaStep:=iParaStep+1;
	  		 ELSIF   	fbReadRegs.bError THEN
	  		 			iParaStep:=999;				
	  		 			iQErrorID:=HITBOT_ERROR.FLT_READ_PARA;					
	  		 END_IF				
 	4://旋转速度比较
				iOldParaStep:=iParaStep;
				IF stLocalPara.stRotateClampPara.rSpeedSet <> stReadPara.rRotateSpeed THEN 
					 iParaStep:=iParaStep + 1;	
				ELSE
					 iParaStep:=iParaStep + 4;
				END_IF
	5://旋转速度赋值
			iOldParaStep:=iParaStep;
			MEMCPY(ADR(arwSetData[1]),ADR(stLocalPara.stRotateClampPara.rSpeedSet),SIZEOF(stLocalPara.stRotateClampPara.rSpeedSet)); 
			arwDataWriteRegs[1]:=arwSetData[2];
			arwDataWriteRegs[2]:=arwSetData[1];
			iParaStep:=iParaStep +1;
	6://旋转角度写入
			 iOldParaStep:=iParaStep;
			 wQuantityWriteRegs:=2;
			 wMBAddWriteRegs:=16#000E;
			 xWriteRegs:=TRUE;
			 IF  fbWriteRegs.bBusy THEN
					 xWriteRegs:=FALSE;
					 iParaStep:=iParaStep+1;
			END_IF	
	7://等待设定完成
				iOldParaStep:=iParaStep;
			 IF  NOT 	fbWriteRegs.bBusy AND  NOT fbWriteRegs.bError THEN
							  iParaStep:=iParaStep +1;
				ELSIF   	fbReadRegs.bError THEN
						 iParaStep:=999;				
						 iQErrorID:=HITBOT_ERROR.FLT_SET_PARA;					
				END_IF	
	8://旋转电流比较
				iOldParaStep:=iParaStep;
				IF stLocalPara.stRotateClampPara.rCurrentSet <> stReadPara.rRotateCurrent THEN 
					 iParaStep:=iParaStep + 1;	
				ELSE
					 iParaStep:=iParaStep + 4;
				END_IF
	9://旋转电流赋值
			iOldParaStep:=iParaStep;
			MEMCPY(ADR(arwSetData[1]),ADR(stLocalPara.stRotateClampPara.rCurrentSet),SIZEOF(stLocalPara.stRotateClampPara.rCurrentSet)); 
			arwDataWriteRegs[1]:=arwSetData[2];
			arwDataWriteRegs[2]:=arwSetData[1];
			iParaStep:=iParaStep +1;
	10://旋转电流写入
			 iOldParaStep:=iParaStep;
			 wQuantityWriteRegs:=2;
			 wMBAddWriteRegs:=16#0010;
			 xWriteRegs:=TRUE;
			 IF  fbWriteRegs.bBusy THEN
					 xWriteRegs:=FALSE;
					 iParaStep:=iParaStep+1;
			END_IF	
	11://等待设定完成
				iOldParaStep:=iParaStep;
			 IF  NOT 	fbWriteRegs.bBusy AND  NOT fbWriteRegs.bError THEN
							  iParaStep:=iParaStep +1;
				ELSIF   	fbReadRegs.bError THEN
						 iParaStep:=999;				
						 iQErrorID:=HITBOT_ERROR.FLT_SET_PARA;					
				END_IF	
	12://写入电机使能
			iOldParaStep:=iParaStep;
			arwDataWriteRegs[1]:=1;
			iParaStep:=iParaStep +1;
	13://开始写入
			 iOldParaStep:=iParaStep;
			 wQuantityWriteRegs:=1;
			 wMBAddWriteRegs:=16#0016;
			 xWriteRegs:=TRUE;
			 IF  fbWriteRegs.bBusy THEN
					 xWriteRegs:=FALSE;
					 iParaStep:=iParaStep+1;
			END_IF	
	14://等待设定完成
				iOldParaStep:=iParaStep;
			 IF  NOT 	fbWriteRegs.bBusy AND  NOT fbWriteRegs.bError THEN
							  iParaStep:=100;
				ELSIF   	fbReadRegs.bError THEN
						 iParaStep:=999;				
						 iQErrorID:=HITBOT_ERROR.FLT_SET_PARA;					
				END_IF	
	100://参数写入完成
				iOldParaStep:=iParaStep;
				iOperType:=stOperType.iWait;
				stPara.xQBusy:=FALSE;
				stPara.xQDone:=TRUE;
				iParaStep:=0;		
	ELSE
		;	
END_CASE
END_ACTION

ACTION ACT_Reset:
IF   xIReset THEN
 
 	 iParaStep:=0;
	 iRunStep:=0;
	 iOldParaStep:=0;
	 iOldRunStep:=0;
	 
	 stPara.xQStart:=FALSE;
	 stPara.xQBusy:=FALSE;
	 stPara.xQError:=FALSE;
 
	 stDevice.xQStart:=FALSE;
	 stDevice.xQBusy:=FALSE;
	 stDevice.xQError:=FALSE;
	 
	 iQErrorID := HITBOT_ERROR.NO_ERROR;
	 xIReset:=FALSE;
END_IF
END_ACTION

ACTION ACT_Running:
IF  NOT  stDevice.xQBusy THEN
 		stDevice.xQRdyCmd:=TRUE;
ELSE
 		stDevice.xQRdyCmd:=FALSE;	
END_IF

CASE  iRunStep OF 
 0://等待开始
 		IF  stDevice.xQStart THEN
		 		stDevice.xQStart:=FALSE;
				stDevice.xQBusy:=TRUE;
				stDevice.xQDone:=FALSE;
				iRunStep:=iRunStep +1;
		END_IF
 1://参数传递
 		 iOldRunStep:=iRunStep;
		 IF iOperType<>stCmdType.iInit THEN
 		 			stPara.xQStart:=TRUE;
					iRunStep:=iRunStep +1;
		 ELSE
				 iRunStep:=iRunStep +2;
		 END_IF
 2://等待参数传递完成
 		 	iOldRunStep:=iRunStep;
 		 IF  stPara.xQDone THEN
				iRunStep:=iRunStep +1;
		 END_IF
 3://开始执行
 		iOldRunStep:=iRunStep;
	  IF 		iOperType=stCmdType.iClamp OR
					iOperType=stCmdType.iRelease THEN
    				iRunStep:=10;
		ELSIF  iOperType=stCmdType.iRotateClamp  OR
					 iOperType=stCmdType.iRotateRelease OR 
					 iOperType=stCmdType.iRotateRelClamp OR 
					 iOperType=stCmdType.iRotateRelRelease THEN
		 				iRunStep:=20;
		ELSIF  		iOperType=stCmdType.iInit  THEN
		 				iRunStep:=30;
		END_IF	
 10://先查询是否已经完成初始化
				iOldRunStep:=iRunStep;
				wMBAddReadRegs:=16#0040;
				wQuantityReadRegs:=1;
				xReadRegs:=TRUE;
				IF  fbReadRegs.bBusy THEN
					xReadRegs:=FALSE;
					iRunStep:=iRunStep+1;
				END_IF
 11://等待读取完成
			 iOldRunStep:=iRunStep;
	  	  IF  NOT 	fbReadRegs.bBusy AND  NOT  	fbReadRegs.bError THEN
				 				//初始化状态反馈
				 				stReadPara.iInitStatus:=arwDataReadRegs[1];
								iRunStep:=iRunStep+1;
	  		 ELSIF   	fbReadRegs.bError THEN
	  		 			iRunStep:=999;				
	  		 			iQErrorID:=HITBOT_ERROR.FLT_READ_PARA;					
	  		 END_IF	
	12://执行完成
	    	iOldRunStep:=iRunStep;
				IF   stReadPara.iInitStatus <>5 THEN
				 			iQErrorID:=HITBOT_ERROR.FLT_NEED_INIT;
							iRunStep:=999;
				ELSE
 							iRunStep:=iRunStep+1;							 
				END_IF
	13://赋值夹持位置
			iOldRunStep:=iRunStep;
			MEMCPY(ADR(arwSetData[1]),ADR(stLocalPara.stClampPara.rPositionSet),SIZEOF(stLocalPara.stClampPara.rPositionSet)); 
			arwDataWriteRegs[1]:=arwSetData[2];
			arwDataWriteRegs[2]:=arwSetData[1];
			iRunStep:=iRunStep +1;

  14://写入夹持位置
			iOldRunStep:=iRunStep;
			wQuantityWriteRegs:=2;
			wMBAddWriteRegs:=16#0002;
			xWriteRegs:=TRUE;
			IF  fbWriteRegs.bBusy THEN
					xWriteRegs:=FALSE;
					iRunStep:=iRunStep+1;
		 END_IF
  15://启动完成
			iOldRunStep:=iRunStep;
			IF  NOT 	fbWriteRegs.bBusy AND  NOT  	fbWriteRegs.bError  THEN
							iRunStep:=iRunStep +1;
			 ELSIF   	fbReadRegs.bError THEN
						iRunStep:=999;				
					  iQErrorID:=HITBOT_ERROR.FLT_RUN_ERROR;					
			 END_IF		
 	16://读取反馈
			 iOldRunStep:=iRunStep;
			 wMBAddReadRegs:=16#0041;
			 wQuantityReadRegs:=8;
			 xReadRegs:=TRUE;
			 IF  fbReadRegs.bBusy THEN
				 xReadRegs:=FALSE;
				 iRunStep:=iRunStep+1;
			 END_IF
 	17://等待读取完成
			 iOldRunStep:=iRunStep;
	  	 IF  NOT 	fbReadRegs.bBusy AND  NOT  	fbReadRegs.bError THEN
				 				//夹持状态反馈
				 				stReadPara.iClampStatus:=arwDataReadRegs[1];
								//夹持位置反馈    
							   
								stReadPara.rFeedBack_ClampPos:=M_Little_Endian(pInputData:=ADR(arwDataReadRegs[2]));
								//夹持速度反馈    
							  
								stReadPara.rFeedBack_ClampSpeed:=M_Little_Endian(pInputData:=ADR(arwDataReadRegs[4]));
								
								//夹持电流反馈
							
								stReadPara.rRotateAngle:=M_Little_Endian(pInputData:=ADR(arwDataReadRegs[6]));
								
								IF   stReadPara.iClampStatus =0 THEN
								 //0-到位
								 			iRunStep:=iRunStep+1;	
								 ELSIF  stReadPara.iClampStatus =1 THEN
									//1-运动中
										  iRunStep:=iRunStep-1;						
								ELSIF  stReadPara.iClampStatus =2 THEN	
								 //2-夹持但未夹取到产品
								 			iRunStep:=iRunStep+1;	
								 			//IF xITryRun THEN//如果空跑状态下夹空不报警
											//			 iRunStep:=iRunStep+1;	 
											//ELSE
											// 		  iRunStep:=999;
											//		  iQErrorID:=HITBOT_ERROR.FLT_CLAMP_EMPTY;		
											//END_IF
								ELSIF   stReadPara.iClampStatus =3 THEN
								 //3-掉落
								 				  iRunStep:=999;
													iQErrorID:=HITBOT_ERROR.FLT_CLAMP_EMPTY;		
								END_IF
	  		 ELSIF   	fbReadRegs.bError THEN
	  		 			iRunStep:=999;				
	  		 			iQErrorID:=HITBOT_ERROR.FLT_READ_PARA;					
	  		 END_IF	
	18://执行完成
	    	iOldRunStep:=iRunStep;
				iRunStep:=100;
				
				
	20://先查询是否已经完成初始化
				iOldRunStep:=iRunStep;
				wMBAddReadRegs:=16#0040;
				wQuantityReadRegs:=1;
				xReadRegs:=TRUE;
				IF  fbReadRegs.bBusy THEN
					xReadRegs:=FALSE;
					iRunStep:=iRunStep+1;
				END_IF
  21://等待读取完成
			 	iOldRunStep:=iRunStep;
	  	  IF  NOT 	fbReadRegs.bBusy AND  NOT  	fbReadRegs.bError THEN
				 				//初始化状态反馈
				 				stReadPara.iInitStatus:=arwDataReadRegs[1];
								iRunStep:=iRunStep+1;
	  		 ELSIF   	fbReadRegs.bError THEN
	  		 			iRunStep:=999;				
	  		 			iQErrorID:=HITBOT_ERROR.FLT_READ_PARA;					
	  		 END_IF	
	22://执行完成
	    	iOldRunStep:=iRunStep;
				IF   stReadPara.iInitStatus <>5 THEN
				 			iQErrorID:=HITBOT_ERROR.FLT_NEED_INIT;
							iRunStep:=999;
				ELSE
 							iRunStep:=iRunStep+1;							 
				END_IF
	23://赋值旋转角度
				iOldRunStep:=iRunStep;
				IF  iOperType=stCmdType.iRotateClamp  OR
					 iOperType=stCmdType.iRotateRelease THEN
							MEMCPY(ADR(arwSetData[1]),ADR(stLocalPara.stRotateClampPara.rPositionSet),SIZEOF(stLocalPara.stRotateClampPara.rPositionSet)); 
							arwDataWriteRegs[1]:=arwSetData[2];
							arwDataWriteRegs[2]:=arwSetData[1];	
							wMBAddWriteRegs:=16#000A;		
						 iRunStep:=iRunStep+1;				
					 
				ELSIF  iOperType=stCmdType.iRotateRelClamp OR 
					 iOperType=stCmdType.iRotateRelRelease THEN
							MEMCPY(ADR(arwSetData[1]),ADR(stLocalPara.stRotateRelAngle),SIZEOF(stLocalPara.stRotateRelAngle)); 
							arwDataWriteRegs[1]:=arwSetData[2];
							arwDataWriteRegs[2]:=arwSetData[1];
							wMBAddWriteRegs:=16#0014;	
						 iRunStep:=iRunStep+1;				
				END_IF  			
	24://写入旋转角度
				iOldRunStep:=iRunStep;
				wQuantityWriteRegs:=2;
				xWriteRegs:=TRUE;
				IF  fbWriteRegs.bBusy THEN
						xWriteRegs:=FALSE;
						iRunStep:=iRunStep+1;
			 END_IF
 	25://启动完成
				iOldRunStep:=iRunStep;
				IF  NOT 	fbWriteRegs.bBusy AND  NOT  	fbWriteRegs.bError  THEN
								iRunStep:=iRunStep +1;
				 ELSIF   	fbReadRegs.bError THEN
							iRunStep:=999;				
						  iQErrorID:=HITBOT_ERROR.FLT_RUN_ERROR;					
				 END_IF		
  26://读取反馈
				iOldRunStep:=iRunStep;
				wMBAddReadRegs:=16#0048;
				wQuantityReadRegs:=8;
				xReadRegs:=TRUE;
				IF  fbReadRegs.bBusy THEN
					xReadRegs:=FALSE;
					iRunStep:=iRunStep+1;
				END_IF
  27://等待读取完成
			 	iOldRunStep:=iRunStep;
	  	  IF  NOT 	fbReadRegs.bBusy AND  NOT  	fbReadRegs.bError THEN
				 				//旋转状态反馈
				 				stReadPara.iRotateStatus:=arwDataReadRegs[1];
								
								//旋转角度反馈         
								stReadPara.rFeedBack_RotatePos:=M_Little_Endian(pInputData:=ADR(arwDataReadRegs[2]));;
							//旋转速度反馈    
						
								stReadPara.rFeedBack_ClampSpeed:=M_Little_Endian(pInputData:=ADR(arwDataReadRegs[4]));;
					  	//旋转电流反馈
								
							  	stReadPara.rFeedBack_RotateCurrent:=M_Little_Endian(pInputData:=ADR(arwDataReadRegs[6]));
								IF    ABS(stReadPara.rFeedBack_RotatePos-stLocalPara.stRotateClampPara.rPositionSet)<2.0 AND 
											 stReadPara.iRotateStatus =0  THEN
								 					iRunStep:=iRunStep+1;	
								END_IF
								IF   stReadPara.iRotateStatus =0 THEN
								 //0-到位
								 			//iRunStep:=iRunStep+1;	
								 ELSIF  stReadPara.iRotateStatus =1  THEN
									//1-运动中
										 // iRunStep:=iRunStep-1;						
								ELSIF  stReadPara.iRotateStatus =2 THEN	
								 //2-堵转
								 
								ELSIF    stReadPara.iRotateStatus =4 THEN
								 //3/这不知道干啥的
								 	// iRunStep:=iRunStep-1;	
								END_IF
	  		 ELSIF   	fbReadRegs.bError THEN
	  		 			iRunStep:=999;				
	  		 			iQErrorID:=HITBOT_ERROR.FLT_READ_PARA;					
	  		 END_IF	
	28://执行完成
	    	iOldRunStep:=iRunStep;
				iRunStep:=100;
  30://初始化
				iOldRunStep:=iRunStep;
				arwDataWriteRegs[1]:=1;//启动
				wQuantityWriteRegs:=1;
				wMBAddWriteRegs:=16#0000;
				xWriteRegs:=TRUE;
				IF  fbWriteRegs.bBusy THEN
						xWriteRegs:=FALSE;
						iRunStep:=iRunStep+1;
			 END_IF
 	31://启动完成
				iOldRunStep:=iRunStep;
				IF  NOT 	fbWriteRegs.bBusy AND  NOT  	fbWriteRegs.bError  THEN
								iRunStep:=iRunStep +1;
				 ELSIF   	fbReadRegs.bError THEN
							iRunStep:=999;				
						  iQErrorID:=HITBOT_ERROR.FLT_RUN_ERROR;					
				 END_IF		
  32://读取反馈
				iOldRunStep:=iRunStep;
				wMBAddReadRegs:=16#0040;
				wQuantityReadRegs:=16;
				xReadRegs:=TRUE;
				IF  fbReadRegs.bBusy THEN
					xReadRegs:=FALSE;
					iRunStep:=iRunStep+1;
				END_IF
  33://等待读取完成
			 	iOldRunStep:=iRunStep;
	  	  IF  NOT 	fbReadRegs.bBusy AND  NOT  	fbReadRegs.bError THEN
				 				//初始化反馈
				 				stReadPara.iInitStatus:=arwDataReadRegs[1];
							//夹持状态反馈         
						  stReadPara.iClampStatus:=arwDataReadRegs[2];		
							//夹持位置反馈       
							stReadPara.rFeedBack_ClampPos:=M_Little_Endian(pInputData:=ADR(arwDataReadRegs[3]));;
							//夹持速度反馈  
							stReadPara.rFeedBack_ClampSpeed:=M_Little_Endian(pInputData:=ADR(arwDataReadRegs[5]));;
							//夹持电流反馈
							stReadPara.rRotateAngle:=M_Little_Endian(pInputData:=ADR(arwDataReadRegs[7]));;
							//旋转状态反馈
				 			stReadPara.iRotateStatus:=arwDataReadRegs[9];
							//旋转角度反馈         
							stReadPara.rFeedBack_RotatePos:=M_Little_Endian(pInputData:=ADR(arwDataReadRegs[10]));
							//旋转速度反馈       
							stReadPara.rFeedBack_ClampSpeed:=M_Little_Endian(pInputData:=ADR(arwDataReadRegs[12]));
							//旋转电流反馈
							stReadPara.rFeedBack_RotateCurrent:=M_Little_Endian(pInputData:=ADR(arwDataReadRegs[14]));
								IF   stReadPara.iInitStatus =5 THEN
								 //5-初始化完成
								 			iRunStep:=iRunStep+1;	
								 ELSIF  stReadPara.iInitStatus =0 THEN
									//0-未初始化		
								ELSE
								 //其他-初始化中
								 	iRunStep:=iRunStep -1;	
								END_IF
	  		 ELSIF   	fbReadRegs.bError THEN
	  		 			iRunStep:=999;				
	  		 			iQErrorID:=HITBOT_ERROR.FLT_READ_PARA;					
	  		 END_IF	
	34://执行完成
	    	iOldRunStep:=iRunStep;
				iRunStep:=100;
 100://运行结束
					stDevice.xQBusy:=FALSE;
					stDevice.xQDone:=TRUE;
					iRunStep:=0;
 END_CASE
 
 
IF  	iOperType=stCmdType.iClamp OR
 			iOperType=stCmdType.iRelease THEN
		ACT_Para_Clamp();
ELSIF  	iOperType=stCmdType.iRotateClamp OR
 			iOperType=stCmdType.iRotateRelease OR
 			iOperType=stCmdType.iRotateRelRelease OR
 			iOperType=stCmdType.iRotateRelClamp THEN
		ACT_Para_Rotate();	 
END_IF
END_ACTION

END_FUNCTION_BLOCK

// ---- POUs/003_FB/0010_LoadCell/FB_Modbus_Tcp.TcPOU
FUNCTION_BLOCK FB_Modbus_Tcp
(*
********************************************************************************
* Name: FB_Modbus_TCP
*
* Author:  Automanh
* Version: 1.0.0
*
* Description:
*   List all modbus TCP Function Block
*
* Remarks:
*
* Revisions:
*   1.0 -AutomanH Rebuild
*********************************************************************************)
VAR_INPUT
END_VAR
VAR_OUTPUT
END_VAR
VAR
 stModbusPara:stModbusPara;
{region "02 :Input status 读取离散量输入相关变量"}
fbReadInputs :FB_MBReadInputs;(*读取离散量输入功能块*)
xReadInputs:BOOL;(*执行条件*)
wQuantityInputs:WORD:=1;(*读取个数*)
wMBAddInputs:WORD:=1;(*读取起始地址*)
arwDataInputs :ARRAY[1..20] OF WORD;(*存放离散量输入的值*)
{endregion}
{region "01:Coil status 读取/写入线圈相关变量"}
fbReadCoils :FB_MBReadCoils;(*读取线圈功能块*)
xReadCoils:BOOL;(*执行条件*)
wQuantityReadCoils:WORD:=1;(*读取个数*)
wMBAddReadCoils:WORD:=1;(*读取起始地址*)
arwDataReadCoils :ARRAY[1..20] OF WORD;(*存放线圈的值*)
	 
			
fbWriteCoils :FB_MBWriteCoils;(*写入线圈功能块*)
xWriteCoils:BOOL;(*执行条件*)
wQuantityWriteCoils:WORD:=1;(*读取个数*)
wMBAddWriteCoils:WORD:=1;(*读取起始地址*)
arwDataWriteCoils :ARRAY[1..20] OF WORD;(*写入线圈的值*)				 
						

fbWriteSingleCoil :FB_MBWriteSingleCoil;(*写入单个线圈功能块*)
xWriteSingleCoil:BOOL;(*执行条件*)
wMBAddWriteSingleCoil:WORD:=1;(*读取起始地址*)
wDataWriteSingleCoil :WORD;(*写入单个线圈的值*)	
{endregion}
{region "04:Input Register 读取输入寄存器相关变量"}	 
fbReadInputRegs :FB_MBReadInputRegs;(*读取输入寄存器功能块*)
xReadInputRegs:BOOL;(*执行条件*)
wQuantityReadInputRegs:WORD:=1;(*读取个数*)
wMBAddReadInputRegs:WORD:=1;(*读取起始地址*)
arwDataReadInputRegs :ARRAY[1..20] OF WORD;(*存放输入寄存器的值*)
{endregion}

{region "03:Holding  Register 读取或写入保存寄存器相关变量"}	 
fbReadRegs :FB_MBReadRegs;(*读取保存寄存器功能块*)
xReadRegs:BOOL;(*执行条件*)
wQuantityReadRegs:WORD:=1;(*读取个数*)
wMBAddReadRegs:WORD:=1;(*读取起始地址*)
arwDataReadRegs :ARRAY[1..20] OF WORD;(*存放保持寄存器的值*)
	 
fbWriteRegs :FB_MBWriteRegs;(*写入保存寄存器功能块*)
xWriteRegs:BOOL;(*执行条件*)
wQuantityWriteRegs:WORD:=1;(*读取个数*)
wMBAddWriteRegs:WORD:=1;(*读取起始地址*)
arwDataWriteRegs :ARRAY[1..20] OF WORD;(*存放保持寄存器的值*)			
				 
		
fbWriteSingleReg :FB_MBWriteSingleReg;(*写入单个保存寄存器功能块*)
xWriteSingleReg:BOOL;(*执行条件*)
wMBAddWriteSingleReg:WORD:=1;(*读取起始地址*)
wDataWriteSingleReg : WORD;(*存放保持寄存器的值*)					
{endregion}
{region "浮点数转化为十进制数 IEEE-754 32位浮点数"}
dwData:DWORD;
rSIGN:LREAL;//符号位
bExponent:BYTE;//指数
bExMemory:BYTE;//记录
dwExponent:DWORD;//指数位
rExponent:LREAL;
rFraction:LREAL;//尾数位	
_xNeedFlag:BOOL;//标记
iMathStep,iMathOldstep:INT;
l_b_repeat:BOOL;
{endregion}
{region "32位单精度浮点数转化为实数"}
ardwData: DWORD;
arwTempData:ARRAY[1..2]OF WORD;
arwInputData:ARRAY[1..2]OF WORD;
{endregion}
{region "实数转化成DWORD"}
rInputRealData:REAL;
{endregion}
END_VAR

METHOD M_Big_Endian : REAL
 VAR_INPUT
 wInputData_1: WORD ;
 wInputData_2: WORD ;
END_VAR
		arwTempData[1]:=	wInputData_1;
		arwTempData[2]:=	wInputData_2;
	  MEMCPY(ADR(M_Big_Endian),ADR(arwTempData[1] ),SIZEOF(M_Big_Endian));
END_METHOD

METHOD M_IEEE754 : REAL
VAR_INPUT
END_VAR
VAR
 E:BYTE;
 M:WORD;
END_VAR
REPEAT
	 l_b_repeat := FALSE;
	 CASE iMathStep OF
		0: //符号位
						
			 IF  dwData.31 =0 THEN
					 rSIGN:=1;
			 ELSIF dwData.31 =1 THEN
					rSIGN:=-1;
			 END_IF
			  l_b_repeat := TRUE;
			 iMathStep:=iMathStep +1;
		1://阶码或指数部分
			 bExponent.7:=dwData.30;
			 bExponent.6:=dwData.29;
			 bExponent.5:=dwData.28;
			 bExponent.4:=dwData.27;
			 bExponent.3:=dwData.26;
			 bExponent.2:=dwData.25;
			 bExponent.1:=dwData.24;
			 bExponent.0:=dwData.23;
			 bExMemory:=bExponent;
			IF  bExMemory>127 THEN
			 		bExponent:=bExMemory-127;
			ELSE
			 		bExponent:=127-bExMemory;
			 END_IF
			 rExponent:=TO_LREAL(EXPT(2,bExponent));
			 l_b_repeat := TRUE;
			 iMathStep:=iMathStep +1;
		2://尾数部分
				IF  dwData.22 THEN
				 		rFraction:=1.0+1*EXPT(2,-1);
				ELSE
				 		rFraction:=1.0;
				END_IF
				IF  dwData.21 THEN
				 		rFraction:=rFraction+1*EXPT(2,-2);
				END_IF
				IF  dwData.20 THEN
				 		rFraction:=rFraction+1*EXPT(2,-3);
				END_IF
				IF  dwData.19 THEN
				 			rFraction:=rFraction+1*EXPT(2,-4);
				END_IF
				IF  dwData.18 THEN
				 			rFraction:=rFraction+1*EXPT(2,-5);
				END_IF
				IF  dwData.17 THEN
				 		rFraction:=rFraction+1*EXPT(2,-6);
				END_IF
				IF  dwData.16 THEN
				 		rFraction:=rFraction+1*EXPT(2,-7);
				END_IF
				IF  dwData.15 THEN
				 			rFraction:=rFraction+1*EXPT(2,-8);
				END_IF
				IF  dwData.14 THEN
				 		rFraction:=rFraction+1*EXPT(2,-9);
				END_IF
				IF  dwData.13 THEN
				 		rFraction:=rFraction+1*EXPT(2,-10);
				END_IF
				IF  dwData.12 THEN
				 			rFraction:=rFraction+1*EXPT(2,-11);
				END_IF
				IF  dwData.11 THEN
				 			rFraction:=rFraction+1*EXPT(2,-12);
				END_IF
				IF  dwData.10 THEN
				 		rFraction:=rFraction+1*EXPT(2,-13);
				END_IF
				IF  dwData.09 THEN
				 		rFraction:=rFraction+1*EXPT(2,-14);
				END_IF
				IF  dwData.08 THEN
				 			rFraction:=rFraction+1*EXPT(2,-15);
				END_IF
				IF  dwData.07 THEN
				 		rFraction:=rFraction+1*EXPT(2,-16);
				END_IF
				IF  dwData.06 THEN
				 		rFraction:=rFraction+1*EXPT(2,-17);
				END_IF
				IF  dwData.05 THEN
				 			rFraction:=rFraction+1*EXPT(2,-18);
				END_IF
				IF  dwData.04 THEN
				 		rFraction:=rFraction+1*EXPT(2,-19);
				END_IF
				IF  dwData.03 THEN
				 		rFraction:=rFraction+1*EXPT(2,-20);
				END_IF
				IF  dwData.02 THEN
				 			rFraction:=rFraction+1*EXPT(2,-21);
				END_IF
				IF  dwData.01 THEN
				 			rFraction:=rFraction+1*EXPT(2,-22);
				END_IF
				IF  dwData.00 THEN
				 		rFraction:=rFraction+1*EXPT(2,-23);
				END_IF
				l_b_repeat := TRUE;
			 	iMathStep:=iMathStep +1;
		3://计算结果
			M_IEEE754:=rSIGN*rExponent*rFraction;
			l_b_repeat := TRUE;
			iMathStep:=999;
	END_CASE
UNTIL l_b_repeat = FALSE
END_REPEAT;
END_METHOD

METHOD M_Little_Endian : REAL
(*
********************************************************************************
* Name: M_Little_Endian
*
* Author:  Automanh
* Version: 1.0.0
*
* Description:
*   Little-Endian Mode
*
*
* Remarks:
*
* Revisions:
*   1.0 -AutomanH Rebuild
*********************************************************************************)
VAR_INPUT
 pInputData:POINTER TO ARRAY[1..2] OF WORD ;
END_VAR
		//MEMCPY(ADR(arwInputData),pInputData,SIZEOF(arwInputData) ); 
	  //arwTempData[1]:=arwInputData[2];
	  //arwTempData[2]:=arwInputData[1];
		arwTempData[1]:=	pInputData^[2];
		arwTempData[2]:=	pInputData^[1];
	  MEMCPY(ADR(M_Little_Endian),ADR(arwTempData[1] ),SIZEOF(M_Little_Endian));
END_METHOD

METHOD M_Modbus : BOOL
VAR_INPUT
END_VAR
{region "02 :Input status 读取离散量输入相关变量"}
fbReadInputs(
	sIPAddr:= stModbusPara.strSlaveIP, 
	nTCPPort:=stModbusPara.iSlavePort , 
	nUnitID:= stModbusPara.bySlaveID, 
	nQuantity:= wQuantityInputs, 
	nMBAddr:= wMBAddInputs, 
	cbLength:=SIZEOF(arwDataInputs) , 
	pDestAddr:=ADR(arwDataInputs) , 
	bExecute:=xReadInputs , 
	tTimeout:=T#1S, 
	bBusy=> , 
	bError=> , 
	nErrId=> , 
	cbRead=> );
{endregion}
	 
{region "01:Coil status 读取/写入线圈相关变量"}
fbReadCoils(
	sIPAddr:= 	stModbusPara.strSlaveIP, 
	nTCPPort:= 	stModbusPara.iSlavePort ,
	nUnitID:= 	stModbusPara.bySlaveID,  
	nQuantity:=wQuantityReadCoils , 
	nMBAddr:=wMBAddReadCoils , 
	cbLength:=SIZEOF(arwDataReadCoils) , 
	pDestAddr:= ADR(arwDataReadCoils), 
	bExecute:= xReadCoils, 
	tTimeout:= T#1S, 
	bBusy=> , 
	bError=> , 
	nErrId=> , 
	cbRead=> );
	 
fbWriteCoils(
	sIPAddr:=	 	stModbusPara.strSlaveIP, 
	nTCPPort:= 	stModbusPara.iSlavePort ,
	nUnitID:= 	stModbusPara.bySlaveID,  
	nQuantity:= wQuantityWriteCoils, 
	nMBAddr:=wMBAddWriteCoils , 
	cbLength:= SIZEOF(arwDataWriteCoils), 
	pSrcAddr:= ADR(arwDataWriteCoils), 
	bExecute:= xWriteCoils, 
	tTimeout:=  T#1S, 
	bBusy=> , 
	bError=> , 
	nErrId=> );		

fbWriteSingleCoil(
	sIPAddr:= 	stModbusPara.strSlaveIP, 
	nTCPPort:= 	stModbusPara.iSlavePort ,
	nUnitID:= 	stModbusPara.bySlaveID,  
	nMBAddr:=wMBAddWriteSingleCoil , 
	nValue:= wDataWriteSingleCoil, 
	bExecute:= xWriteSingleCoil, 
	tTimeout:= T#1S, 
	bBusy=> , 
	bError=> , 
	nErrId=> );
{endregion}
{region "04:Input Register 读取输入寄存器相关变量"}	
 fbReadInputRegs(
	sIPAddr:= 	stModbusPara.strSlaveIP,  
	nTCPPort:= 	stModbusPara.iSlavePort , 
	nUnitID:= 	stModbusPara.bySlaveID,   
	nQuantity:=wQuantityReadInputRegs , 
	nMBAddr:= wMBAddReadInputRegs, 
	cbLength:= SIZEOF(arwDataReadInputRegs), 
	pDestAddr:=ADR(arwDataReadInputRegs) , 
	bExecute:=xReadInputRegs , 
	tTimeout:=  T#1S, 
	bBusy=> , 
	bError=> , 
	nErrId=> , 
	cbRead=> );
		 
{endregion}
	 
{region "03:Holding  Register 读取或写入保存寄存器相关变量"}	 
fbReadRegs(
	sIPAddr:= 	stModbusPara.strSlaveIP, 
	nTCPPort:= 	stModbusPara.iSlavePort ,
	nUnitID:= 	stModbusPara.bySlaveID,  
	nQuantity:= wQuantityReadRegs, 
	nMBAddr:= wMBAddReadRegs, 
	cbLength:= SIZEOF(arwDataReadRegs), 
	pDestAddr:=ADR(arwDataReadRegs) , 
	bExecute:= xReadRegs, 
	tTimeout:= T#1S, 
	bBusy=> , 
	bError=> , 
	nErrId=> , 
	cbRead=> );
		 
fbWriteRegs(
	sIPAddr:= 	stModbusPara.strSlaveIP, 
	nTCPPort:= 	stModbusPara.iSlavePort ,
	nUnitID:= 	stModbusPara.bySlaveID,  
	nQuantity:=wQuantityWriteRegs , 
	nMBAddr:=wMBAddWriteRegs , 
	cbLength:= SIZEOF(arwDataWriteRegs), 
	pSrcAddr:=ADR(arwDataWriteRegs) , 
	bExecute:=xWriteRegs , 
	tTimeout:=  T#1S, 
	bBusy=> , 
	bError=> , 
	nErrId=> );
		 
fbWriteSingleReg(
	sIPAddr:= 	stModbusPara.strSlaveIP,  
	nTCPPort:= 	stModbusPara.iSlavePort , 
	nUnitID:= 	stModbusPara.bySlaveID,   
	nMBAddr:= wMBAddWriteSingleReg, 
	nValue:=wDataWriteSingleReg , 
	bExecute:=xWriteSingleReg , 
	tTimeout:=  T#1S, 
	bBusy=> , 
	bError=> , 
	nErrId=> );	 		
{endregion}
END_METHOD

METHOD M_RealToWord : ARRAY[1..2] OF WORD
VAR_INPUT
END_VAR
MEMCPY(ADR(arwTempData[1]),ADR(rInputRealData),SIZEOF(arwTempData) ); 
M_RealToWord[1]:=arwTempData[2];
M_RealToWord[2]:=arwTempData[1];
END_METHOD

END_FUNCTION_BLOCK

// ---- POUs/003_FB/0002_Camera/FB_Camera.TcPOU
FUNCTION_BLOCK FB_Camera
(*
********************************************************************************
* Name: FB_Camera
*
* Author:  AutomanH
* Version: 1.0.0
*
* Description:
*	Camera trigger and camera lights control
*
* Remarks:
*
*
* Revisions:
*   V1.0.0 -Automanh 2022.06.08
*		V2.0.0-Automanh 2022.07.15 add Timeout Error and xQDone Single
*********************************************************************************)
VAR_INPUT
	xlInit	:BOOL;(*初始化*)
	xlTrigger:BOOL;(*相机触发*)
	xlTriggerHmi:BOOL;(*触摸屏相机触发*)
	xlLight  :BOOL;(*是否存在光源*)
	xlReady	 :BOOL;(*相机准备就绪信号*)
	xlAutoMode:BOOL;(*自动模式*)
	xlManualMode:BOOL;(*手动模式*)
	xITryRun:BOOL;(*空跑*)
	tlDelay: TIME;  (*打开光源与拍照间隔的时间*)
	xIDeviceRunning :BOOL;(*单循环运行*)
	
END_VAR
VAR_OUTPUT
	xQStart	:BOOL;			//开始拍照
	xQLight: BOOL := FALSE;//打开光源
	xQCompleted:BOOL;		//拍照完成
	xQAlarm	: BOOL := FALSE;// 报警输出
	xQBusy	 	:BOOL;
	xQHmiAlarm	:STRING;//报警输出
	xQDone	  :BOOL;
END_VAR
VAR_IN_OUT
	ilCompleted :INT;(*拍照完成*)
END_VAR
VAR
	bStep:BYTE;
	{attribute 'hide'}
	tonDelay: TON;//计时器
	{attribute 'hide'}
	tonAlarmTime :Ton;//报警计时器
	{attribute 'hide'}
	tTimeout:TON;
END_VAR

ACT_Init();
ACT_Trigger();
ACT_Alarm();

ACTION ACT_Alarm:
IF NOT xlReady THEN
	xQHmiAlarm:='Not Ready';
ELSIF xlReady AND NOT xQBusy THEN
 	xQHmiAlarm:='Ready';
ELSIF xQAlarm THEN
	xQHmiAlarm:='Time out';
END_IF
END_ACTION

ACTION ACT_Init:
IF  xlInit THEN
	xlTrigger:=FALSE;	
	xlTriggerHmi:=FALSE;
	xlLight :=FALSE;
	ilCompleted:=0;
	xQStart:=FALSE;
	xQLight:=FALSE;
	xQCompleted:=FALSE;
	xQAlarm	  :=FALSE;
	xQBusy    :=FALSE;
	xQDone		:=FALSE;
	xlInit	  :=FALSE;
END_IF
END_ACTION

ACTION ACT_Trigger:

CASE bStep OF
	0://等待触发
		tonDelay(IN:=FALSE);
		tonAlarmTime(IN:=FALSE);
		ilCompleted:=0;
		IF (( (xlAutomode OR xIDeviceRunning) AND xlTrigger) OR
				(xlManualmode AND xlTriggerHmi)) AND (xlReady OR xITryRun) THEN
			xlTrigger:=xlTriggerHmi:=FALSE;
			xQCompleted:=FALSE;
			xQBusy:=TRUE;
			xQDone:=FALSE;
			bStep:=bStep +1;
		END_IF
	
	1://打开光源信号
		 IF  NOT xITryRun THEN
			 IF xlLight THEN
				 xQLight:=TRUE;
			 END_IF
		 END_IF
			 bStep:=bStep+1;		
	2://开始拍照
		IF  NOT   xITryRun THEN
			 tonDelay(IN:=TRUE,PT:=tlDelay,	Q=>,ET=>);
			 IF  tonDelay.Q  THEN
				 xQStart:=TRUE;
				 xQHmiAlarm:='Started';
				 tonDelay(IN:=FALSE);
				 bStep:=bStep+1;		
			 END_IF
		ELSE
				bStep:=bStep+1;		
		END_IF
 3://拍照结束
	 		IF  ilCompleted = 1 OR xITryRun THEN 
			 	ilCompleted:=0;
			 	xQStart:=FALSE;
				xQLight:=FALSE;
				bStep:=bStep+1;	
				xQCompleted:=TRUE;	
			ELSE
				tonAlarmTime(IN:=TRUE,PT:=T#3S,	Q=>,ET=>);
				IF    tonAlarmTime.Q THEN
				 	xQStart:=FALSE;
					xQLight:=FALSE;
					xQAlarm:=TRUE;
					tonAlarmTime(IN:=FALSE);
					bStep:=0;	
				END_IF
			END_IF
	4://关闭光源
			xQCompleted:=TRUE;
			xQLight:=FALSE;
			bStep:=bStep+1;	
	5://流程结束
			xQHmiAlarm:='Completed';
			xQBusy:=FALSE;
			xQDone:=TRUE;
			bStep:=0;	
END_CASE
END_ACTION

END_FUNCTION_BLOCK

// ---- POUs/001_Station/S08_MainLine.TcPOU
PROGRAM S08_MainLine
VAR
	//工站
	station					: REFERENCE TO FB_Station:=fbstation[8];
	//伺服
	fbMainLineAxis	 :REFERENCE TO FB_Axis:=fbAxis[15];	//	主流线伺服

	
	//延时
	arTonDelay :ARRAY[1..20] OF TON;
	//返回值
	UdiReturnValue :ARRAY[1..20] OF UDINT;
	//清除过程记录
	xClearProcessStatus	:BOOL;

	i: INT;
	bCounter:INT;//环形线计数
	// 临时变量
	_xFirstCycle: BOOL;
	//过程记录
	tsModuleProcess:ARRAY[1..gc_ModuleProNo] OF DUT_Process;
	xClearModuleProcessDone:BOOL;
	bClearProcessStep	:BYTE;
	// //环形线尾端传感器
	xMainLineEndCheckSensor: ARRAY[1..2] OF BOOL;
	NextPosR_TRIG:R_TRIG;
	// 计算周长步骤
	wActionCalibration: WORD;
	// 起始位置
	rStartPoition: REAL;
	// 结束位置
	rEndPoition: REAL;
	DataEmptyR_TRIG:R_TRIG;
	CounterR_TRIG:R_TRIG;
	CycleCounter:INT;//环形线周期次数
	testR_TRIG:Tc2_Standard.R_TRIG;
	// 测试使用待删
	xtest: BOOL;
END_VAR

A_Input();
Alarm();
Delay();
FlowAuto();
FlowInit();
General();
ILC();
TipAuto();
TipManual();
Z_Output();

ACTION A_Input:
//传感器
xMainLineEndCheckSensor[1] :=IxLineEndSensor1Reached;
xMainLineEndCheckSensor[2] :=IxLineEndSensor2Reached;
END_ACTION

ACTION Alarm:
//
station.adwAlarm[1].00:=station.xInitTimeout;	  			//S08Label 初始化超时
station.adwAlarm[1].01	:=	fbMainLineAxis.xError	;//	S08主流线旋转伺服报错
station.adwAlarm[1].02	:=	fbMainLineAxis.xNotPowerOn	;//	S08主流线旋转伺服未使能
station.adwAlarm[1].03	:=	fbMainLineAxis.xMoveTimeout	;//	S08主流线旋转伺服移动超时
(*station.adwAlarm[1].04	:=	TRUE;//	S08主流线有残余产品*)
END_ACTION

ACTION Delay:
arTonDelay[01](IN:= , PT:=T#0.1S , Q=> , ET=> );
(*arTonDelay[02](IN:=  , PT:=T#1S , Q=> , ET=> );*)//自动程序用
arTonDelay[03](IN:=   , PT:=T#1S , Q=> , ET=> );
arTonDelay[04](IN:= , PT:=T#0.1S , Q=> , ET=> );
arTonDelay[05](IN:= , PT:=T#0.1S , Q=> , ET=> );
arTonDelay[06](IN:= , PT:=T#0.1S , Q=> , ET=> );
arTonDelay[07](IN:= , PT:=T#0.1S , Q=> , ET=> );
arTonDelay[08](IN:= , PT:=T#0.1S , Q=> , ET=> );
arTonDelay[09](IN:= , PT:=T#0.1S , Q=> , ET=> );
arTonDelay[10](IN:= NOT fbMainLineAxis.xbusy , PT:=T#0.1S , Q=> , ET=> );//TipAuto使用
END_ACTION

ACTION FlowAuto:

//-----------------------------------------初始化是否完成判断----------------------------------------------
IF NOT station.xInitDone 
THEN
 	station.iStepAuto:=0;
 	station.xDone:=FALSE;
	station.xRunningOffProhibit := FALSE ;//运行中信号Off禁止
ELSIF station.xRunning  OR   tsModuleProcess[1].xProcessStarted
THEN
//-----------------------------------------动作步骤--------------------------------------------------------
CASE station.iStepAuto OF	  
	0: //----Home Step，等待启动----
		IF station.xDisabled 
			AND station.xCanRun 
			AND NOT fbMachine[1].xStopped 
			AND NOT station.xSingleRunning 
		THEN
			station.xDone:=TRUE;
		END_IF
		
		IF  station.xSingleRunning 
			OR station.xCanRun 
			//AND NOT station.xDone 
			AND NOT station.xDisabled 
			AND NOT fbMachine[1].xStopped
		THEN
			station.xCycleEnable:=TRUE;
			//station.xDone:= FALSE;  
			station.iStepAuto:= 10;
		END_IF
    10: //复位数据 
				 FOR i:=1 TO gc_ModuleProNo BY 1 DO
						 MEMSET(ADR(tsModuleProcess[i]),0,SIZEOF(tsModuleProcess[i]));
				 END_FOR
			station.iStepAuto:=50;
			
	50://等待各个工位完成信号
		IF  S01_Loading.station.xDone  		AND 
			S02_LidInjecting.station.xDone  AND 
			S03_LidChecking.station.xDone 	AND 
			S04_AluCovering.station.xDone  		AND 
			S05_Adjusting.station.xDone  AND 
			S06_Cutting.station.xDone 	AND 
			xS07MainlineRunPermit 	THEN 
			station.iStepAuto:=60;
		END_IF
	55://不允许各工位操作
			Station.xDone:=FALSE;//不允许操作
			 station.iStepAuto:=60;	
	60://读取原点偏移量
		 IF NOT _xFirstCycle THEN
		   stData.Axis[15].rMovePosition[2] := stData.Axis[15].rMovePosition[1] ;
		   _xFirstCycle := TRUE ;
		 END_IF
		   station.iStepAuto:=80;	
		   
//	70:////Restore_after_Estop_Process1 皮带线移动流程
//			IF tsModuleProcess[1].xProcessNotStarted AND NOT  tsModuleProcess[1].xProcessStarted THEN
//					station.iStepAuto :=80; (*process not started*)
//			ELSIF  tsModuleProcess[1].xProcessStarted AND NOT  tsModuleProcess[1].xProcessCompleted THEN
//				 station.iStepAuto := 90;(*process started*)
//			ELSIF  tsModuleProcess[1].xProcessCompleted AND NOT tsModuleProcess[1].xQDataCompleted  THEN
//					station.iStepAuto := 150 ;(*process completed*)
//			ELSIF tsModuleProcess[1].xQDataCompleted THEN
//					station.iStepAuto :=160;(*Qdata completed *)
//			ELSE
//					station.iStepAuto :=80; 
//			END_IF		  
	80://储存当前位置
			tsModuleProcess[1].xProcessNotStarted:=TRUE;
			stData.Axis[15].rMovePosition[3]:=fbMainLineAxis.rActPos;
			station.iStepAuto:=100;
//	90://判断伺服位置是否合理
//			IF      ( ABS(stData.Axis[15].rMovePosition[3]+stData.Axis[15].rRelativeDistance))+0.1>=ABS(stData.Axis[15].rMovePosition[2]) AND 
//					  ( ABS(stData.Axis[15].rMovePosition[3]+stData.Axis[15].rRelativeDistance))-0.1<=ABS(stData.Axis[15].rMovePosition[2]) THEN
//					  station.iStepAuto:=110;(*伺服已经移动过了*)
//			ELSIF  ABS(stData.Axis[15].rMovePosition[3])+0.1>=ABS(stData.Axis[15].rMovePosition[2]) AND 
//				   ABS(stData.Axis[15].rMovePosition[3])-0.1<=ABS(stData.Axis[15].rMovePosition[2]) THEN
//				     station.iStepAuto:=100;(*伺服需要移动*)
//			END_IF
	100://数据更新 位置
		tsModuleProcess[1].xProcessStarted:=TRUE;
		stData.Axis[15].rMovePosition[2] := stData.Axis[15].rMovePosition[2] +stData.Axis[15].rRelativeDistance ;
		arTonDelay[02](IN:= FALSE , PT:=T#50MS , Q=> , ET=> );
	   	station.iStepAuto:= 110;
	
	110:
	 	 arTonDelay[02](IN:= TRUE , PT:=T#50MS , Q=> , ET=> );
		   IF arTonDelay[02].Q THEN
       		station.iStepAuto:=130;
					arTonDelay[02](IN:=FALSE, PT:=T#50MS , Q=> , ET=> );
       END_IF
	130:
			fbMainLineAxis.xMoveAuto[2]:=TRUE;
			IF fbMainLineAxis.xMoveInPos[2] THEN
				station.iStepAuto :=140; 
			END_IF		
	140://计数
				bCounter:= bCounter +1;
				station.iStepAuto :=145; 
	145://检查是否需要回原点
				station.iStepAuto :=150; 	
	150://数据传递
				FOR  i:= 40 TO 1 BY -1 DO
					MEMCPY(ADR(arMainlineFixtureData[i+2]),ADR(arMainlineFixtureData[i]),SIZEOF(arMainlineFixtureData[i]));
				END_FOR
			tsModuleProcess[1].xQDataCompleted:=TRUE;
			 station.iStepAuto:=160;
	160://判断产品状态
	  	 FOR i:= 1 TO gc_MainLineFixtureNumber BY 1 DO 
					 IF 	arMainLineFixtureData[i].stProduct.xLoading_OK AND 
						  arMainLineFixtureData[i].stProduct.xlidInjecting_OK AND
						  arMainLineFixtureData[i].stProduct.xLidChecking_OK AND 
						  arMainLineFixtureData[i].stProduct.xAluCovering_OK AND 
						  arMainLineFixtureData[i].stProduct.xAdjusting_OK    AND
						  arMainLineFixtureData[i].stProduct.xCutting_OK  THEN
					   		arMainLineFixtureData[i].stProduct.xALL_OK := TRUE ;
							arMainLineFixtureData[i].stProduct.xPart_Normal := FALSE ;
							arMainLineFixtureData[i].stProduct.xPart_NG := FALSE ;
					ELSIF	
							arMainLineFixtureData[i].stProduct.xLoading_NOK OR 
						  arMainLineFixtureData[i].stProduct.xlidInjecting_NOK OR
						  arMainLineFixtureData[i].stProduct.xLidChecking_NOK OR 
						  arMainLineFixtureData[i].stProduct.xAluCovering_NOK OR 
						  arMainLineFixtureData[i].stProduct.xAdjusting_NOK    OR
						  arMainLineFixtureData[i].stProduct.xCutting_NOK  THEN
							arMainLineFixtureData[i].stProduct.xALL_OK := FALSE ;
							arMainLineFixtureData[i].stProduct.xPart_Normal := FALSE ;
							arMainLineFixtureData[i].stProduct.xPart_NG := TRUE ;
					ELSE
							arMainLineFixtureData[i].stProduct.xALL_OK := FALSE ;
							arMainLineFixtureData[i].stProduct.xPart_Normal := TRUE ;
							arMainLineFixtureData[i].stProduct.xPart_NG := FALSE ;
					 END_IF
				
				//以下待删
					arMainLineFixtureData[i].stProduct.xALL_OK := TRUE ;
			  	arMainLineFixtureData[i].stProduct.xPart_Normal := FALSE ;
	      	arMainLineFixtureData[i].stProduct.xPart_NG := FALSE ;
        END_FOR	
		 station.iStepAuto:=170;	
			
	170://清除各站的过程记录
			xClearProcessStatus:=TRUE;
			IF S02_LidInjecting.xClearModuleProcessDone 	 AND 
				S03_LidChecking.xClearModuleProcessDone 	AND 
				S04_AluCovering.xClearModuleProcessDone  	AND 
				S05_Adjusting.xClearModuleProcessDone  		AND 
				S06_Cutting.xClearModuleProcessDone 	    THEN 
					station.iStepAuto:=180;
			END_IF
	180://过程记录清除完成
			xClearProcessStatus:=FALSE;
			IF 	NOT S02_LidInjecting.xClearModuleProcessDone 	 AND 
				NOT S03_LidChecking.xClearModuleProcessDone 	AND 
				NOT S04_AluCovering.xClearModuleProcessDone  	AND 
				NOT S05_Adjusting.xClearModuleProcessDone  		AND 
				NOT S06_Cutting.xClearModuleProcessDone 	THEN 
						station.iStepAuto:=190;
			END_IF
	190://启动各个工位
			FOR  i:= 1 TO 6 BY 1 DO 
				fbStation[i].xDone:=FALSE;
			END_FOR
			xS07MainlineRunPermit:=FALSE;
			station.iStepAuto:=500;	
	500://清除本站过程记录及数据
			FOR i:=1 TO gc_ModuleProNo BY 1 DO
				MEMSET(ADR(tsModuleProcess[i]),0,SIZEOF(tsModuleProcess[i]));
			END_FOR
		
			 station.iStepAuto:=999;
	999://----Single Run Finish----
			
		station.iStepAuto :=0;
		IF NOT station.xSingleContinuousRun THEN
			station.xSingleRunFlag:=FALSE;
		END_IF
		station.xCycleEnable:=FALSE;	
		station.xDone:=TRUE;
		
		
		
		
1000://回原点流程
				tsModuleProcess[2].xProcessCompleted:=TRUE;
				fbMainLineAxis.xReferenceAuto := TRUE ;
				station.iStepAuto:=1010;	
1010://伺服回原点完成
	IF  fbAxisHome[15].home_done THEN 
		 	fbMainLineAxis.xReferenceAuto  := FALSE ;
		 	station.iStepAuto:=1050;	
	END_IF
1050://回原点完成
				tsModuleProcess[2].xProcessCompleted:=TRUE;
				_xFirstCycle:=FALSE;
				bCounter:=1;	
				station.iStepAuto:=142;	
		
		
	ELSE
		;	
END_CASE



END_IF
END_ACTION

ACTION FlowInit:
IF NOT station.xIniting THEN
  station.iStepInit:=0;    
ELSE
//--------------------------------------------初始化步序----------------------------------
CASE station.iStepInit OF	
 0://  
  	IF station.xIniting THEN	
  	  station.iStepInit:=10;	
  	END_IF	
10://复位数据
		 bCounter:=1;
		_xFirstCycle:=FALSE;
		FOR i:=1 TO gc_ModuleProNo BY 1 DO
				MEMSET(ADR(tsModuleProcess[i]),0,SIZEOF(tsModuleProcess[i]));
			END_FOR
		station.iStepInit:=20;
20://伺服上电
	fbMainLineAxis.xPowerInit:=TRUE;
	IF  fbMainLineAxis.xPowerOn THEN
			station.iStepInit:=30;
	END_IF
30://等待其他设备初始化完成
			IF  S01_Loading.station.xInitDone  		AND 
			S02_LidInjecting.station.xInitDone  AND 
			S03_LidChecking.station.xInitDone 	AND 
			S04_AluCovering.station.xInitDone  		AND 
			S05_Adjusting.station.xInitDone  AND 
			S06_Cutting.station.xInitDone 	AND 
			S07_BoxCarrying.station.xInitDone 	THEN
			station.iStepInit:=35;
		END_IF
35://传感器检测
		IF   IxS01Sensor1Reached  OR
			  IxS01Sensor2Reached  OR
			  IxS02Sensor1Reached  OR
			  IxS02Sensor2Reached  OR  
			//  IxS04Sensor1Reached  OR
			//  IxS04Sensor2Reached  OR
			  IxLineEndSensor1Reached OR
			  IxLineEndSensor2Reached OR	
        IxLineEndCheckSensor1	 OR
        IxLineEndCheckSensor2	THEN
			  	station.adwAlarm[1].04	:=	TRUE;//	S08主流线有残余产品,请检查
		ELSE
		 		station.iStepInit:=40;	
		END_IF
40://皮带回原点
		fbMainLineAxis.xReferenceAuto := TRUE ;
	   	station.iStepInit:=50;
50://回原点完成
	IF  fbAxisHome[15].home_done THEN 
		 fbMainLineAxis.xReferenceAuto  := FALSE ;
		 station.iStepInit:=60;  
	END_IF
55:	//旋转伺服上电
	fbMainLineAxis.xPowerInit:=TRUE;
	IF  fbMainLineAxis.xPowerOn THEN
		station.iStepInit :=60;
	END_IF
			
60://伺服到待机点
     fbMainLineAxis.xMoveAuto[1] := TRUE ;
	IF fbMainLineAxis.xMoveInPos[1] THEN 
       station.iStepInit:=100;	
	END_IF
100://清除数据
	FOR  i:=1 TO gc_MainLineFixtureNumber BY 1DO
		MEMSET(ADR(arMainlineFixtureData),0,SIZEOF(arMainlineFixtureData));
	END_FOR
  station.iStepInit:=999;	
999://初始化完成	
	station.iStepInit:=0;
	station.xInitDone:=TRUE;  
END_CASE
END_IF
END_ACTION

ACTION General:
{region "主流线上各个工位的位置"}
//S01
arCurFixtureNumStation[1]:=1;
arCurFixtureNumStation[2]:=2;
//S02
arCurFixtureNumStation[3]:=11;
arCurFixtureNumStation[4]:=12;
//s03
arCurFixtureNumStation[5]:=17;
arCurFixtureNumStation[6]:=18;
arCurFixtureNumStation[7]:=19;
arCurFixtureNumStation[8]:=20;
arCurFixtureNumStation[9]:=21;
//s04
arCurFixtureNumStation[10]:=29;
arCurFixtureNumStation[11]:=30;
//s05
arCurFixtureNumStation[12]:=31;
arCurFixtureNumStation[13]:=32;
//S06
arCurFixtureNumStation[14]:=33;
arCurFixtureNumStation[15]:=34;
arCurFixtureNumStation[16]:=35;
//尾端
arCurFixtureNumStation[17]:=41;
arCurFixtureNumStation[18]:=42;
{endregion}
//////去下一个位置
NextPosR_TRIG(CLK:= fbMachine[1].xManualMode AND fbMainLineAxis.xMoveHmi[6], Q=> );
IF  NextPosR_TRIG.Q THEN
 stData.Axis[15].rMovePosition[6]:=fbMainLineAxis.rActPos +fbMainLineAxis.rRelativeDistance;
END_IF

{region "计算环形线周长程序"}
CASE wActionCalibration OF   
  10://回原点
  fbMainLineAxis.xReferenceAuto:= TRUE ;
  	wActionCalibration:=15;
  15:
	 IF  fbAxisHome[15].home_done THEN 
		 fbMainLineAxis.xReferenceAuto  := FALSE ;
		wActionCalibration:=100;
	 END_IF
  20://Jog正向，遇到原点传感器停止
   stData.Axis[15].rJogVelocity :=0.1;  
	fbMainLineAxis.xJogForwardAuto := TRUE ;
	 IF  arAxisSensorH[15] THEN 
		 fbMainLineAxis.xJogForwardAuto := FALSE ; 
			wActionCalibration:=30;
			rStartPoition:=fbMainLineAxis.rActPos;
	 END_IF 
  60: //高速走定位，理论值前10MM处停止
	stData.Axis[15].rMovePosition[5] :=(9191*5)-10; 
	wActionCalibration:=70;
	
70:
	fbMainLineAxis.xMoveAuto[5] := TRUE ;
	 IF fbMainLineAxis.xMoveInPos[5] THEN 
	 fbMainLineAxis.xMoveAuto[5] := FALSE ; 
	 wActionCalibration:=80;
	 END_IF 
80:
	  stData.Axis[15].rJogVelocity :=0.1;  
	fbMainLineAxis.xJogForwardAuto := TRUE ;
 IF   arAxisSensorH[15] THEN 
	 fbMainLineAxis.xJogForwardAuto := FALSE ; 
 		wActionCalibration:=90;
		rEndPoition:=fbMainLineAxis.rActPos;
 END_IF 
90:
	stData.Axis[15].rRelativeDistance:=((rEndPoition-rStartPoition)/450)*2;
		wActionCalibration:=0;
END_CASE    
{endregion}
{region '计算主流线一周的次数'}
CounterR_TRIG(CLK:= arAxisSensorH[15] , Q=> );
	IF  CounterR_TRIG.Q THEN
			CycleCounter:=bCounter-CycleCounter;
	END_IF
	 
{endregion}
{region '测试使用'}
testR_TRIG(CLK:=xtest , Q=> );
IF  	 testR_TRIG.Q THEN
			FOR  i:= 40 TO 1 BY -1 DO
					MEMCPY(ADR(arMainlineFixtureData[i+2]),ADR(arMainlineFixtureData[i]),SIZEOF(arMainlineFixtureData[i]));
					IF i=1 THEN
					EXIT;		
					END_IF
				END_FOR
END_IF
{endregion}
END_ACTION

ACTION ILC:

//---------------------------------------------------工站可执行-------------------------------------------------------
station.xCanRun :=TRUE ;

//---------------------------------------------------气缸动作条件-------------------------------------------


//---------------------------------------------------伺服动作条件-------------------------------------------

fbMainLineAxis.xRunILC := 
fbMainLineAxis.xMoveILC[1] :=
fbMainLineAxis.xMoveILC[2] :=
fbMainLineAxis.xMoveILC[3] :=
fbMainLineAxis.xMoveILC[4] :=
fbMainLineAxis.xMoveILC[5] := 
fbMainLineAxis.xMoveILC[6] := 
		S01_Loading.fbVTCCyl_1.xHP_Delay AND 
		S01_Loading.fbVTCCyl_2.xHP_Delay AND 
		S02_LidInjecting.fbHOZAdjustCyl_1.xHP_Delay AND
		//S02_LidInjecting.fbHOZAdjustCyl_2.xHP_Delay AND
		S02_LidInjecting.fbHOZAdjustCyl_3.xHP_Delay AND
		//	S02_LidInjecting.fbHOZAdjustCyl_4.xHP_Delay AND
		S03_LidChecking.fbHOZAdjustCyl_1.xHP_Delay   AND
		S03_LidChecking.fbHOZAdjustCyl_2.xHP_Delay   AND
		S03_LidChecking.fbHOZAdjustCyl_3.xHP_Delay   AND
		S03_LidChecking.fbHOZAdjustCyl_4.xHP_Delay   AND
		S03_LidChecking.fbHOZAdjustCyl_5.xHP_Delay   AND
		S03_LidChecking.fbHOZAdjustCyl_6.xHP_Delay   AND
		S03_LidChecking.fbHOZAdjustCyl_7.xHP_Delay   AND	
		S03_LidChecking.fbHOZAdjustCyl_8.xHP_Delay   AND
		S04_AluCovering.fbZAxisMove_1.xMoveInPos[1] AND 
		S04_AluCovering.fbZAxisMove_2.xMoveInPos[1] AND
		S04_AluCovering.fbHOZAdjustCyl_1.xHP_Delay AND
	//	S04_AluCovering.fbHOZAdjustCyl_2.xHP_Delay AND
		S04_AluCovering.fbHOZAdjustCyl_3.xHP_Delay AND
	//	S04_AluCovering.fbHOZAdjustCyl_4.xHP_Delay AND
		S05_Adjusting.fbZAxisMove_1.xMoveInPos[1] AND 
		S05_Adjusting.fbZAxisMove_2.xMoveInPos[1] AND
		S06_Cutting.fbVTCAdjustCyl.xHP_Delay AND
		S06_Cutting.fbHOZCyl.xHP_Delay AND
		S06_Cutting.fbHOZReachedCyl_1.xHP_Delay AND
		S06_Cutting.fbHOZReachedCyl_2.xHP_Delay AND
		S06_Cutting.fbVTCCyl.xHP_Delay AND
		S06_Cutting.fbPressCyl_1.xHP_Delay AND
		S06_Cutting.fbPressCyl_2.xHP_Delay ;
END_ACTION

ACTION TipAuto:

//------------------------------------------------AutoTip Cylinder--------------------------------
	
//------------------------------------------------AutoTip Servo--------------------------------
//**************************************
FOR i:= 1 TO 5 BY 1 DO 
	IF fbMainLineAxis.xMoveAuto[i] THEN
		fbMainLineAxis.iPosNumber := i ;
	END_IF
	
END_FOR


IF  fbMachine[1].xAutoMode AND NOT fbMachine[1].xRunning AND arTonDelay[10].Q   THEN
	IF	fbMainLineAxis.iPosNumber=1 	AND NOT fbMainLineAxis.xMoveInPos[1] THEN 	station.adwAutoTip[1].10:=TRUE	;	END_IF//轴伺服自动时位置不在位置1
	IF	fbMainLineAxis.iPosNumber=2	AND NOT fbMainLineAxis.xMoveInPos[2]	THEN 	station.adwAutoTip[1].11:=TRUE	;	END_IF//轴伺服自动时位置不在位置2
	IF	fbMainLineAxis.iPosNumber=3	AND NOT fbMainLineAxis.xMoveInPos[3]	THEN 	station.adwAutoTip[1].12:=TRUE	;	END_IF//轴伺服自动时位置不在位置3
	IF	fbMainLineAxis.iPosNumber=4	AND NOT fbMainLineAxis.xMoveInPos[4]	THEN 	station.adwAutoTip[1].13:=TRUE	;	END_IF//轴伺服自动时位置不在位置4
	IF	fbMainLineAxis.iPosNumber=5	AND NOT fbMainLineAxis.xMoveInPos[5]	THEN 	station.adwAutoTip[1].14:=TRUE	;	END_IF//轴伺服自动时位置不在位置5
END_IF
END_ACTION

ACTION TipManual:
//--------------------------------------------ManualTip------------------------------------------------------

//-------------------------------------------气缸提示---------------------------------------------------------




/////////////////////////////////////////////////////////////////////////////////////////////////////////////////
END_ACTION

ACTION Z_Output:
(**************************气缸输出********************************)
END_ACTION

END_PROGRAM

// ---- POUs/001_Station/S02_LidInjecting.TcPOU
PROGRAM S02_LidInjecting
VAR
	//工站
	station					: REFERENCE TO FB_Station:=fbstation[2];
	//气缸
	fbHOZAdjustCyl_1	:REFERENCE TO FB_Cylinder:=fbCylinder[7];	//	上层水平调整气缸1
//	fbHOZAdjustCyl_2	:REFERENCE TO FB_Cylinder:=fbCylinder[8];	//	上层水平调整气缸2
	fbHOZAdjustCyl_3	:REFERENCE TO FB_Cylinder:=fbCylinder[9];	//	下层水平调整气缸1
//	fbHOZAdjustCyl_4	:REFERENCE TO FB_Cylinder:=fbCylinder[10];	//	下层水平调整气缸2
	fbROTCyl	:REFERENCE TO FB_Cylinder:=fbCylinder[11];	//	旋转气缸-防滴液
	//伺服
	fbXAxisMove	 :REFERENCE TO FB_Axis:=fbAxis[3];	//	注液工位X轴伺服
	fbYAxisMove	 :REFERENCE TO FB_Axis:=fbAxis[4];	//	注液工位Y轴伺服
	fbZAxisMove	 :REFERENCE TO FB_Axis:=fbAxis[5];	//	注液工位Z轴伺服
	fbStirAxis	 :REFERENCE TO FB_Axis:=fbAxis[9];	//	磁珠搅拌
	//蠕动泵
	(*直接用全局变量*)
	//称
	fbMKC204C:REFERENCE TO FB_MT_MKC:=fbMCK204w;
	//自动校准
	fbAutoCalib	:REFERENCE TO FB_AutoCal:=fbAutoCal;
	//压力传感器

	//延时
	arTonDelay :ARRAY[1..20] OF TON;
	//返回值
	UdiReturnValue :ARRAY[1..20] OF UDINT;
	//本地过程数据
	arProcessDataStation : ARRAY [1..2] OF DUT_MainlineFixture;
	i: INT;
	xNeedCalibration: BOOL;
	// 蠕动泵校准完成
	xCalibCompleted: BOOL;
	// X轴循环
	bXCounter: BYTE;
	//过程记录
	tsModuleProcess:ARRAY[1..gc_ModuleProNo] OF DUT_Process;
	xClearModuleProcessDone:BOOL;
	bClearProcessStep	:BYTE;
	// //首次循环
	_FirstCycle: ARRAY[1..10] OF BOOL;
	//深孔板到位传感器
	xSensorReached:ARRAY[1..2] OF BOOL;
	// 蠕动泵控制器个数
	bPumpControllerCounter: BYTE;
	// 校准延时定时器
	tSteadyTimer: TON;
	//蠕动泵排空使用
	RudongPump_R_TRIG:ARRAY[1..2] OF R_TRIG;
	// 排空液体步骤
	iRudongPumpEmptyStep,iRudongPumpEmptyOldStep: INT;
	//排空液体超时
	tEmptyTimeOut:TON;
	// 校准注液次数
	_InjectCounuter: INT;
	//校准注液的实际液量
	arrMckDisplay:ARRAY[1..10] OF REAL;
	//校准超时
	tCalibrationTimeOut:TON;
	//校准步骤
	iCalibStep:INT;
	tMCalibTimeOut:TON;
	//标志位
	arxPushBusy:ARRAY[1..12] OF BOOL;
	// 临时变量
	arrVolume: ARRAY[1..2] OF REAL;
	arrTest:ARRAY[1..10] OF REAL;
	rTEST:REAL;
		// 压力传感器读取步骤
	iRepeatLoadCellStep,iOldRepeatLoadCellStep: INT;
	arxLoadCellBusy:ARRAY[1..6] OF BOOL;
	tLoadCellDelay:TON;
	tLoadCellTimeout:TON;
	//VBA表格使用的变量
	arrVBARecordData:ARRAY[1..50] OF REAL;
	iEasyPumpController:INT;
	iEasyPumpGHead:INT;
	iCycleCounter:INT;
	iBackAngle:INT;
	rAccuracySet:REAL;
	rSetVolume:REAL;
	rRunTime:REAL;
	


	// //泵头类型
	iPumpType: INT;
	// //软管类型
	iSoftType: INT;
	//泵头类型
	iPumpHeadType: INT;
	//校准次数
	iCalibCounter:INT;
END_VAR

A_Input();
Alarm();
Delay();
FlowAuto();
FlowInit();
General();
ILC();
TipAuto();
TipManual();
Z_Output();
ACT_test();

ACTION A_Input:
//气缸

fbHOZAdjustCyl_1.xWP_Sensor	:=	IxS02HOZAdjustCyl_1WP  AND IxS02HOZAdjustCyl_2WP	;
fbHOZAdjustCyl_1.xHP_Sensor	:=	IxS02HOZAdjustCyl_1HP	 AND IxS02HOZAdjustCyl_2HP;
fbHOZAdjustCyl_3.xWP_Sensor	:=	IxS02HOZAdjustCyl_3WP	AND IxS02HOZAdjustCyl_4WP	;
fbHOZAdjustCyl_3.xHP_Sensor	:=	IxS02HOZAdjustCyl_3HP	AND IxS02HOZAdjustCyl_4HP;;
fbROTCyl.xWP_Sensor	:=	IxS02ROTCylWP	;
fbROTCyl.xHP_Sensor	:=	IxS02ROTCylHP	;

xSensorReached[1]:=IxS02Sensor1Reached	;//	注液工位¶到位传感器1
xSensorReached[2]:=IxS02Sensor2Reached	;//	注液工位¶到位传感器2
END_ACTION

ACTION ACT_test:

CASE stManualCalib.iMCalibStep OF
 0://等待按键
		IF  stManualCalib.xStart  AND
			  stManualCalib.iPumpContorller>=1 AND 
				stManualCalib.iPumpContorller<=12 AND 
				stManualCalib.iPumpModule>=1 AND 
				stManualCalib.iPumpModule<=9 THEN
			  stManualCalib.xModulePushStart:=FALSE;		 
				stManualCalib.xModulePushOK:=FALSE;			
				stManualCalib.xCalibTestStart:=FALSE;				 
				stManualCalib.xCalibTestOK:=FALSE;						
				stManualCalib.xRecordDataStart:=FALSE;	
				stManualCalib.xRecordDataOK:=FALSE;						 
				stManualCalib.xStart  :=FALSE;
				stManualCalib.xBusy  :=TRUE;
				stManualCalib.xDone :=FALSE;	 
				stManualCalib.iMCalibStep:=stManualCalib.iMCalibStep +1;
		ELSIF   stManualCalib.xGotoPosition THEN
		 		stManualCalib.iMCalibStep:=50;
		END_IF
1://参数赋值
	 	stManualCalib.iOldMCalibStep:=stManualCalib.iMCalibStep;
		stData.EasyPumps[stManualCalib.iPumpContorller].rCalFluVolume:=stManualCalib.rSetVolume;
		stData.EasyPumps[stManualCalib.iPumpContorller].iModuleAdress:=stManualCalib.iPumpModule;
		stData.EasyPumps[stManualCalib.iPumpContorller].rCalTime:=stManualCalib.rRunTime;
		//stData.EasyPumps[stManualCalib.iPumpContorller].rCalNum:=stManualCalib.iCycleNum;
		stData.EasyPumps[stManualCalib.iPumpContorller].rModuleRealFluVolume:=stManualCalib.rAverageRealVolume;
		stData.EasyPumps[stManualCalib.iPumpContorller].rCalBackAngle:=stManualCalib.iBackAngle;
		stManualCalib.iMCalibStep:=stManualCalib.iMCalibStep +1;
2://写入校准参数
	 	stManualCalib.iOldMCalibStep:=stManualCalib.iMCalibStep;
		stManualCalib.iMCalibStep:=stManualCalib.iMCalibStep +1;	
3://等待写入完成
	 	stManualCalib.iOldMCalibStep:=stManualCalib.iMCalibStep;
	  stManualCalib.xModulePushStart:=TRUE;
		stManualCalib.xModulePushOK:=FALSE;
		stManualCalib.xNeedInjectAgain:=FALSE;
		stManualCalib.iMCalibStep:=stManualCalib.iMCalibStep +1;	
4://清除原有数据
	 	stManualCalib.iOldMCalibStep:=stManualCalib.iMCalibStep;
		MEMSET(ADR(stManualCalib.arrRealVolume[1]),0,SIZEOF(stManualCalib.arrRealVolume));
		stManualCalib.rAverageRealVolume:=0; 
		stManualCalib.iInjectCounter:=1;
	 	stManualCalib.iMCalibStep:=stManualCalib.iMCalibStep +1;	
5://检查
		IF   stManualCalib.xModulePushStart THEN
			stData.EasyPumps[stManualCalib.iPumpContorller].rCalNum:=6;	//连续注液六次	
		ELSIF    stManualCalib.xCalibTestStart THEN
		 	stData.EasyPumps[stManualCalib.iPumpContorller].rCalNum:=1;	//连续注液两次
		ELSIF   stManualCalib.xRecordDataStart THEN
			stData.EasyPumps[stManualCalib.iPumpContorller].rCalNum:=1;	//注液一次
		END_IF  
		stManualCalib.iMCalibStep:=stManualCalib.iMCalibStep +1;	
6://称清零
	 	stManualCalib.iOldMCalibStep:=stManualCalib.iMCalibStep;
	  fbMCK.stDeviceOpe.xClearZeroInstanly_HMI:=TRUE;
		IF fbMCK.xQBusy THEN
							 stManualCalib.iMCalibStep:=stManualCalib.iMCalibStep +1;	
		END_IF
7://等待清零完成
	 	stManualCalib.iOldMCalibStep:=stManualCalib.iMCalibStep;
	  IF  fbMCK.xQDone THEN
			  	stManualCalib.iMCalibStep:=stManualCalib.iMCalibStep +1;
		 ELSIF  fbMCK.xQError THEN
				  fbMCK.xIReset:=TRUE;
					stManualCalib.iMCalibStep:=6;	
		 END_IF
8://开始单通道注液
	 	stManualCalib.iOldMCalibStep:=stManualCalib.iMCalibStep;
	  fbEasyPumps[stManualCalib.iPumpContorller].stDeviceOpe.xModulePush_Auto:=TRUE;
		IF  fbEasyPumps[stManualCalib.iPumpContorller].xQBusy THEN
				stManualCalib.iMCalibStep:=stManualCalib.iMCalibStep +1;	
		END_IF
9://等待注液完成
	 	stManualCalib.iOldMCalibStep:=stManualCalib.iMCalibStep;
	 	stManualCalib.tStableDelay(IN:= FALSE);
	 	IF  fbEasyPumps[stManualCalib.iPumpContorller].xQDone THEN
				stManualCalib.iMCalibStep:=stManualCalib.iMCalibStep +1;	
		END_IF
10://等待
					 stManualCalib.tStableDelay(IN:= TRUE, PT:=T#6S , Q=> , ET=> );
					 IF  stManualCalib.tStableDelay.Q THEN
									stManualCalib.tStableDelay(IN:= FALSE);
									stManualCalib.iMCalibStep:=stManualCalib.iMCalibStep +1;	
					 END_IF			 
11://读取称的读数
	 	stManualCalib.iOldMCalibStep:=stManualCalib.iMCalibStep;
	 	fbMCK.stDeviceOpe.xAcquireWeight_RealTime_HMI:=TRUE;
		IF fbMCK.xQBusy THEN
					stManualCalib.iMCalibStep:=stManualCalib.iMCalibStep +1;	
		END_IF
12://等待完成
	 	stManualCalib.iOldMCalibStep:=stManualCalib.iMCalibStep;
	  IF  fbMCK.xQDone THEN
				IF  (fbMCK.stParOut.rCurrentWeight <=stManualCalib.rSetVolume*0.1 )THEN
										stManualCalib.iMCalibStep:=6;
				ELSE
							IF  stManualCalib.xModulePushStart   THEN
									stManualCalib.arrRealVolume[stManualCalib.iInjectCounter]:=fbMCK.stParOut.rCurrentWeight;
							ELSIF  stManualCalib.xCalibTestStart THEN
								 stManualCalib.arrRealVolume[stManualCalib.iCalibCounter]:=fbMCK.stParOut.rCurrentWeight;	
							ELSIF  stManualCalib.xRecordDataStart THEN
									stManualCalib.arrRecordVolume[stManualCalib.iRecordCounter]:=fbMCK.stParOut.rCurrentWeight;
							END_IF
			  			stManualCalib.iMCalibStep:=stManualCalib.iMCalibStep +1;	
					END_IF
		 ELSIF  fbMCK.xQError THEN
				  fbMCK.xIReset:=TRUE;
					 stManualCalib.iMCalibStep:=6;
		 END_IF
13://注液计数
	 	stManualCalib.iOldMCalibStep:=stManualCalib.iMCalibStep;
	 	IF  stManualCalib.xModulePushStart THEN
	  			stManualCalib.iInjectCounter := stManualCalib.iInjectCounter +1;
		ELSIF   stManualCalib.xCalibTestStart THEN
				 	stManualCalib.iCalibCounter := stManualCalib.iCalibCounter +1;
		ELSIF  stManualCalib.xRecordDataStart THEN
						stManualCalib.iRecordCounter := stManualCalib.iRecordCounter +1;
		END_IF
	 	stManualCalib.iMCalibStep:=stManualCalib.iMCalibStep +1;	
14://
	 	stManualCalib.iOldMCalibStep:=stManualCalib.iMCalibStep;
	 	IF   stManualCalib.xModulePushStart THEN
				IF 	 stManualCalib.iInjectCounter >1 THEN
							stManualCalib.iMCalibStep:=stManualCalib.iMCalibStep +1;
				ELSE
							stManualCalib.iMCalibStep:=6;
				END_IF
		ELSIF   stManualCalib.xCalibTestStart THEN
				IF 	 stManualCalib.iCalibCounter >3 THEN
							stManualCalib.iMCalibStep:=stManualCalib.iMCalibStep +1;
				ELSE
							stManualCalib.iMCalibStep:=6;
				END_IF
		ELSIF   stManualCalib.xRecordDataStart THEN
				IF 	 stManualCalib.iRecordCounter >50 THEN
							stManualCalib.iMCalibStep:=stManualCalib.iMCalibStep +1;
				ELSE
							stManualCalib.iMCalibStep:=6;
				END_IF			 
		END_IF
			 
15://计算平均液量或者校准的精度
	 	stManualCalib.iOldMCalibStep:=stManualCalib.iMCalibStep;
		IF  stManualCalib.xModulePushStart THEN
						stManualCalib.rAverageRealVolume:=stManualCalib.arrRealVolume[1]/6; 
						stManualCalib.rESVolume:=(stManualCalib.rAverageRealVolume-stManualCalib.rSetVolume)/stManualCalib.rSetVolume;//偏差值
						IF  ABS( stManualCalib.rESVolume)>stData.EasyPumps[stManualCalib.iPumpContorller].iAccuracySet*0.7 THEN
						 		stManualCalib.xNeedInjectAgain:=TRUE;
						END_IF
								stManualCalib.xModulePushStart:=FALSE;
								stManualCalib.xModulePushOK:=TRUE;
								stManualCalib.iMCalibStep:=stManualCalib.iMCalibStep +1;
		 ELSIF  stManualCalib.xCalibTestStart THEN
									stManualCalib.rESVolume:=FC_BubbleSort_Max(i_i_Counter:=3 , i_arrReal:= stManualCalib.arrRealVolume);//最大值
									stManualCalib.rEIVolume:=FC_BubbleSort_Min(i_i_Counter:=3, i_arrReal:= stManualCalib.arrRealVolume);//最小值
									stManualCalib.rESVolume:=(stManualCalib.rESVolume-stManualCalib.rSetVolume)/stManualCalib.rSetVolume;//上偏差
									stManualCalib.rEIVolume:=(stManualCalib.rEIVolume-stManualCalib.rSetVolume)/stManualCalib.rSetVolume;//下偏差	 
									 IF  stManualCalib.rESVolume>stData.EasyPumps[stManualCalib.iPumpContorller].iAccuracySet*0.9  OR 
											 	stManualCalib.rEIVolume<-1*stData.EasyPumps[stManualCalib.iPumpContorller].iAccuracySet*0.9 	THEN
													 	FOR i:=1 TO 3 BY 1 DO
																stManualCalib.rAverageRealVolume:=stManualCalib.rAverageRealVolume +stManualCalib.arrRealVolume[i];
														END_FOR
														 stManualCalib.rAverageRealVolume:=stManualCalib.rAverageRealVolume/3;
													 stManualCalib.xCalibTestStart:=FALSE;
													 stManualCalib.xCalibTestOK:=FALSE;
													 stManualCalib.iMCalibStep:=stManualCalib.iMCalibStep +1;
											//	//如果上下偏差不均衡  我们需要进行微调处理
										  // IF  ABS(ABS( stManualCalib.rESVolume)-ABS(stManualCalib.rEIVolume))<=stData.EasyPumps[stManualCalib.iPumpContorller].iAccuracySet*0.5 THEN
											//		 stManualCalib.iMCalibStep:=stManualCalib.iMCalibStep +1;
											// ELSE
											//		  stManualCalib.iMCalibStep:=stManualCalib.iMCalibStep +3;
											// END_IF
									 ELSE
													 stManualCalib.xCalibTestStart:=FALSE;
													 stManualCalib.xCalibTestOK:=TRUE;
													 stManualCalib.xRecordDataStart:=TRUE;
													 stManualCalib.xRecordDataOK:=FALSE;
													 stManualCalib.iRecordCounter:=1;
													 stManualCalib.iMCalibStep:=4;
									 END_IF
			ELSIF stManualCalib.xRecordDataStart THEN
											stManualCalib.xRecordDataStart:=FALSE;
											stManualCalib.xRecordDataOK:=TRUE;	
											 stManualCalib.xBusy  :=FALSE;
											 stManualCalib.xDone  :=TRUE;	 
											 stManualCalib.iMCalibStep:=0;			
		  END_IF
16://写入校准参数
	 	stManualCalib.iOldMCalibStep:=stManualCalib.iMCalibStep;
				stData.EasyPumps[stManualCalib.iPumpContorller].rModuleRealFluVolume:=stManualCalib.rAverageRealVolume;
				fbEasyPumps[stManualCalib.iPumpContorller].stDeviceOpe.xCalibAction_Hmi:=TRUE;
				IF  fbEasyPumps[stManualCalib.iPumpContorller].xQBusy THEN
							stManualCalib.iMCalibStep:=stManualCalib.iMCalibStep +1;	
				END_IF
17://等待写入完成
	 	stManualCalib.iOldMCalibStep:=stManualCalib.iMCalibStep;
	 	IF  fbEasyPumps[stManualCalib.iPumpContorller].xQDone THEN
				stManualCalib.xCalibTestStart:=TRUE;
				stManualCalib.iCalibCounter:=1;
					stManualCalib.iMCalibStep:=20;	
		END_IF	
	
18://开始微调
	 	stManualCalib.iOldMCalibStep:=stManualCalib.iMCalibStep;
		fbEasyPumps[stManualCalib.iPumpContorller].stDeviceOpe.xAdjust_Hmi:=TRUE;
		IF  fbEasyPumps[stManualCalib.iPumpContorller].xQBusy THEN
				stManualCalib.iMCalibStep:=stManualCalib.iMCalibStep +1;	
		END_IF
19://等待写入完成
	 	stManualCalib.iOldMCalibStep:=stManualCalib.iMCalibStep;
	 	IF  fbEasyPumps[stManualCalib.iPumpContorller].xQDone THEN
		 		stManualCalib.xCalibTestStart:=TRUE;
				stManualCalib.iMCalibStep:=20;	
		END_IF
20://校准结束,开始测试校准效果
			IF  stManualCalib.xNeedInjectAgain THEN
			 	stManualCalib.iMCalibStep:=1;
			ELSE
			 	stManualCalib.iMCalibStep:=4;
			END_IF
50://伺服上电
			 fbXAxisMove.xPowerInit := TRUE ;
			 fbYAxisMove.xPowerInit := TRUE ;
			 fbZAxisMove.xPowerInit := TRUE ;
			IF fbXAxisMove.xPowerOn AND   fbYAxisMove.xPowerOn AND  fbZAxisMove.xPowerOn THEN 
						stManualCalib.iMCalibStep:=stManualCalib.iMCalibStep +1;	
			END_IF	
51://停止蠕动泵
		 FOR i:=1 TO  12 BY 1 DO
						fbEasyPumps[i].stDeviceOpe.xStop_Hmi:=TRUE;
						IF  fbEasyPumps[i].xQBusy THEN
						 		arxPushBusy[i]:=TRUE;
						END_IF
		 END_FOR
		 	FOR   i :=1 TO 12 BY  1  DO
			 			IF NOT  arxPushBusy[i] THEN
						 		EXIT;
						ELSIF i =12 THEN
						 	  stManualCalib.iMCalibStep:=stManualCalib.iMCalibStep +1;	
					  END_IF
			END_FOR

52://等待蠕动泵全部停止
				 IF   		fbEasyPumps[1].xQDone AND
									fbEasyPumps[2].xQDone AND
									fbEasyPumps[3].xQDone AND
								  fbEasyPumps[4].xQDone AND
									fbEasyPumps[5].xQDone AND
									fbEasyPumps[6].xQDone AND
									fbEasyPumps[7].xQDone AND
								  fbEasyPumps[8].xQDone AND
									fbEasyPumps[9].xQDone AND
									fbEasyPumps[10].xQDone AND
									fbEasyPumps[11].xQDone AND
								  fbEasyPumps[12].xQDone THEN						
								  stManualCalib.iMCalibStep:=stManualCalib.iMCalibStep +1;		
					 END_IF;	

53://Z轴伺服上升
		fbZAxisMove.xMoveAuto[1]:=TRUE;
		IF fbZAxisMove.xMoveInPos[1]   THEN
			  stManualCalib.iMCalibStep:=stManualCalib.iMCalibStep +1;	
		END_IF	
54://防滴液气缸回原
	fbROTCyl.xInit:=TRUE;
	IF fbROTCyl.xHP_Delay THEN
		station.iStepInit :=50;
	END_IF

55://XY轴回参考位
		fbXAxisMove.xMoveAuto[1]:=TRUE;
		fbYAxisMove.xMoveAuto[1]:=TRUE;
		IF fbXAxisMove.xMoveInPos[1]  AND fbYAxisMove.xMoveInPos[1]  THEN
			station.iStepInit:=90;	
		END_IF
					
			
 END_CASE
END_ACTION

ACTION Alarm:
station.adwAlarm[1].00	:=	station.xInitTimeout	;//	S02 初始化超时
//station.adwAlarm[1].01	:=	fbRudongPump[1].xError	;//	S02注液工位蠕动泵1报错
//station.adwAlarm[1].02	:=	fbRudongPump[2].xError	;//	S02注液工位蠕动泵2报错
//station.adwAlarm[1].03	:=	fbRudongPump[3].xError	;//	S02注液工位蠕动泵3报错
//station.adwAlarm[1].04	:=	fbRudongPump[4].xError	;//	S02注液工位蠕动泵4报错
//station.adwAlarm[1].05	:=	fbRudongPump[5].xError	;//	S02注液工位蠕动泵5报错
//station.adwAlarm[1].06	:=	fbRudongPump[6].xError	;//	S02注液工位蠕动泵6报错
//station.adwAlarm[1].07	:=	fbRudongPump[7].xError	;//	S02注液工位蠕动泵7报错
//station.adwAlarm[1].08	:=	fbRudongPump[8].xError	;//	S02注液工位蠕动泵8报错
//station.adwAlarm[1].09	:=	fbRudongPump[9].xError	;//	S02注液工位蠕动泵9报错
//station.adwAlarm[1].10	:=	fbRudongPump[10].xError	;//	S02注液工位蠕动泵10报错
//station.adwAlarm[1].11	:=	fbRudongPump[11].xError	;//	S02注液工位蠕动泵11报错
//station.adwAlarm[1].12	:=	fbRudongPump[12].xError	;//	S02注液工位蠕动泵12报错
station.adwAlarm[1].13	:=	fbHOZAdjustCyl_1.xHP_Off 	;//	S02上层水平调整气缸1原点未到位
station.adwAlarm[1].14	:=	fbHOZAdjustCyl_1.xWP_Off 	;//	S02上层水平调整气缸1动点未到位
station.adwAlarm[1].15	:=	fbHOZAdjustCyl_3.xHP_Off	;//	S02下层水平调整气缸1原点未到位
station.adwAlarm[1].16	:=	fbHOZAdjustCyl_3.xWP_Off	;//	S02下层水平调整气缸1动点未到位
station.adwAlarm[1].17	:=	fbROTCyl.xHP_Off	;//	S02防滴液旋转气缸原点未到位
station.adwAlarm[1].18	:=	fbROTCyl.xWP_Off	;//	S02防滴液旋转气缸动点未到位
station.adwAlarm[1].19	:=	fbXAxisMove.xError	;//	S02注液工位X轴伺服报错
station.adwAlarm[1].20	:=	fbXAxisMove.xNotPowerOn	;//	S02注液工位X轴伺服未使能
station.adwAlarm[1].21	:=	fbXAxisMove.xMoveTimeout	;//	S02注液工位X轴伺服移动超时
station.adwAlarm[1].22	:=	fbYAxisMove.xError	;//	S02注液工位Y轴伺服报错
station.adwAlarm[1].23	:=	fbYAxisMove.xNotPowerOn	;//	S02注液工位Y轴伺服未使能
station.adwAlarm[1].24	:=	fbYAxisMove.xMoveTimeout	;//	S02注液工位Y轴伺服移动超时
station.adwAlarm[1].25	:=	fbZAxisMove.xError	;//	S02注液工位Z轴伺服报错
station.adwAlarm[1].26	:=	fbZAxisMove.xNotPowerOn	;//	S02注液工位Z轴伺服未使能
station.adwAlarm[1].27	:=	fbZAxisMove.xMoveTimeout	;//	S02注液工位Z轴伺服移动超时
//station.adwAlarm[1].28	:=	fbStirAxis.xError	;//	S02注液工位搅拌旋转伺服报错
//station.adwAlarm[1].29	:=	fbStirAxis.xNotPowerOn	;//	S02注液工位搅拌旋转伺服未使能
//station.adwAlarm[1].30	:=	fbStirAxis.xMoveTimeout	;//	S02注液工位搅拌旋转伺服移动超时
station.adwAlarm[1].31	:=	fbMKC204C.xError	;//	S03注液工位称重设备报警

(*station.adwAlarm[2].0	:=	TRUE	;//S03注液工位排空超时.*)

	//station.adwAlarm[2].01	:=	TRUE	;//	S02注液工位1号桶液量不足，请更换母液
	//station.adwAlarm[2].02	:=	TRUE	;//	S02注液工位2号桶液量不足，请更换母液
	//station.adwAlarm[2].03	:=	TRUE	;//	S02注液工位3号桶液量不足，请更换母液
	//station.adwAlarm[2].04	:=	TRUE	;//	S02注液工位4号桶液量不足，请更换母液
	//station.adwAlarm[2].05	:=	TRUE	;//	S02注液工位5号桶液量不足，请更换母液
  //station.adwAlarm[2].06	:=	TRUE	;//	S02注液工位6号桶液量不足，请更换母液
	//station.adwAlarm[2].07	:=	TRUE	;//	S02注液工位压力传感器读取超时报警，请检查
END_ACTION

ACTION Delay:

